# B&R Automation Studio project CombinedLinenSoiledA9KAN (part 15)

#### _actInterfaceApplication.st
```iecst
(********************************************************************
 * COPYRIGHT -- Herbert Kannegiesser GmbH
 ********************************************************************
 * Program: mnParam
 * File: _actInterfaceApplication.st
 * Author: hunholz
 * Created: March 28, 2012
 ********************************************************************
 * Implementation of program mnParam
 ********************************************************************)

(* Kommando-Interface zur Applikation über IFmnParam *)
ACTION _actInterfaceApplication:

	CASE _PmIntern.enCycIfState OF

		cs_IfIdle:

			//*************************************************
			// Kein Applikations-Befehl aktiv. Warte auf Befehl
			//*************************************************

			CASE IFmnParam.In.Edit.wCommand OF

				MNPARAM_CMD_NOCOMMAND:

					IFmnParam.Out.Edit.wStatus := MNPARAM_STAT_NOCOMMAND;

				MNPARAM_CMD_FILLEDITOR:

					IF _xAllowCommands THEN

						_xAllowCommands := FALSE;

						// Warten bis das Füllen des Editors abgeschlossen ist.
						_PmIntern.enCycIfState := cs_IfFillEditor;

						IFmnParam.Out.Edit.wStatus := KG_CMDSTAT_BUSY;

						// Füllen des Editors starten
						_PmIntern.enCycFillEditor := cs_feStart;

					ELSE

						// Kommando ablehnen
						IFmnParam.Out.Edit.wStatus := KG_CMDSTAT_NOTREADY;
						// Kommando muss zurückgenommen werden
						_PmIntern.enCycIfState := cs_IfReady;

					END_IF

				MNPARAM_CMD_SAVEEDITOR:

					IF _xAllowCommands THEN

						_xAllowCommands := FALSE;

						// Warten bis das Sichern des Editors abgeschlossen ist
						_PmIntern.enCycIfState := cs_IfSaveEditor;

						IFmnParam.Out.Edit.wStatus := KG_CMDSTAT_BUSY;

						_LogEntryIn.wErrorNo := _MNPARAM_LOG_STARTSAVE;
						_InsertRB(wPtrStart := _wPtrRBstart, wPtrRead := _wPtrRBread, wPtrWrite := _wPtrRBwrite);

						// Sichern starten
						_PmIntern.enCycSaveEditor := cs_seStart;

					ELSE

						// Kommando ablehnen
						IFmnParam.Out.Edit.wStatus := KG_CMDSTAT_NOTREADY;
						// Kommando muss zurückgenommen werden
						_PmIntern.enCycIfState := cs_IfReady;

					END_IF

				MNPARAM_CMD_CREATE_INDCONT:

					IF _xAllowCommands THEN

						_xAllowCommands := FALSE;

						// Warten bis das Anlegen einer Instanz abgeschlossen ist
						_PmIntern.enCycIfState := cs_IfCreateIndCont;

						IFmnParam.Out.Edit.wStatus := KG_CMDSTAT_BUSY;

						// Parameter übernehmen
						_wCreateCont := IFmnParam.In.Edit.bContainer;
						_wCreateInst := IFmnParam.In.Edit.wContainerInstance;

						_LogEntryIn.wErrorNo := _MNPARAM_LOG_STARTCREATE;
						_LogEntryIn.lAttr1 := _wCreateCont;
						_LogEntryIn.lAttr2 := _wCreateInst;
						_InsertRB(wPtrStart := _wPtrRBstart, wPtrRead := _wPtrRBread, wPtrWrite := _wPtrRBwrite);

						// Instanz anlegen
						_PmIntern.enCycCreate := cs_CrtStart;

					ELSE

						// Kommando ablehnen
						IFmnParam.Out.Edit.wStatus := KG_CMDSTAT_NOTREADY;
						// Kommando muss zurückgenommen werden
						_PmIntern.enCycIfState := cs_IfReady;

					END_IF

				MNPARAM_CMD_DELETE_INDCONT:

					IF _xAllowCommands THEN

						_xAllowCommands := FALSE;

						// Warten bis das Löschen der Instanz abgeschlossen ist
						_PmIntern.enCycIfState := cs_IfDeleteIndCont;

						IFmnParam.Out.Edit.wStatus := KG_CMDSTAT_BUSY;

						// Parameter übernehmen
						_wDelCont := IFmnParam.In.Edit.bContainer;
						_wDelInst := IFmnParam.In.Edit.wContainerInstance;

						_LogEntryIn.wErrorNo := _MNPARAM_LOG_STARTDELETE;
						_LogEntryIn.lAttr1 := _wDelCont;
						_LogEntryIn.lAttr2 := _wDelInst;
						_InsertRB(wPtrStart := _wPtrRBstart, wPtrRead := _wPtrRBread, wPtrWrite := _wPtrRBwrite);

						// Löschen starten
						_PmIntern.enCycDelState := cs_DelStart;

					ELSE

						// Kommando ablehnen
						IFmnParam.Out.Edit.wStatus := KG_CMDSTAT_NOTREADY;
						// Kommando muss zurückgenommen werden
						_PmIntern.enCycIfState := cs_IfReady;

					END_IF

				MNPARAM_CMD_COPY_INDCONT:

					IF _xAllowCommands THEN

						_xAllowCommands := FALSE;

						// Warten bis das Kopieren der Instanz abgeschlossen ist
						_PmIntern.enCycIfState := cs_IfCopyIndCont;

						IFmnParam.Out.Edit.wStatus := KG_CMDSTAT_BUSY;

						// Parameter übernehmen
						_wCopyCont := IFmnParam.In.Edit.bContainer;
						_wCopyInst := IFmnParam.In.Edit.wContainerInstance;
						_wCopyInstFrom := IFmnParam.In.Edit.wContainerInstanceFrom;

						_LogEntryIn.wErrorNo := _MNPARAM_LOG_STARTCOPY;
						_LogEntryIn.lAttr1 := _wCopyCont;
						_LogEntryIn.lAttr2 := _wCopyInst;
						_InsertRB(wPtrStart := _wPtrRBstart, wPtrRead := _wPtrRBread, wPtrWrite := _wPtrRBwrite);

						// Kopieren starten
						_PmIntern.enCycCopy := cs_CpyStart;

					ELSE

						// Kommando ablehnen
						IFmnParam.Out.Edit.wStatus := KG_CMDSTAT_NOTREADY;
						// Kommando muss zurückgenommen werden
						_PmIntern.enCycIfState := cs_IfReady;

					END_IF

				MNPARAM_CMD_BACKUP:

					IF _xAllowCommands THEN

						_xAllowCommands := FALSE;

						// USB-Flashdisk muss gesteckt sein
						IF IFmnSystem.Out.xUSBStickReady THEN

							// Warten bis Backup beendet ist
							_PmIntern.enCycIfState := cs_IfBackup;

							IFmnParam.Out.Edit.wStatus := KG_CMDSTAT_BUSY;

							_LogEntryIn.wErrorNo := _MNPARAM_LOG_STARTBACKUP;
							_LogEntryIn.lAttr1 := 0;
							_LogEntryIn.lAttr2 := 0;
							_InsertRB(wPtrStart := _wPtrRBstart, wPtrRead := _wPtrRBread, wPtrWrite := _wPtrRBwrite);

							// Devicenamen der USB-Flashdisk übernehmen
							_sUSBInterface := IFmnSystem.Out.sInterfaceUSB;

							// Backup starten
							_PmIntern.enCycBackup := cs_BacUSBlinkDevice;

						ELSE

							// Es ist keine USB-Flashdisk gesteckt
							IFmnParam.Out.Edit.wStatus := MNPARAM_STAT_NOUSBSTICK;
							// Kommando muss zurückgenommen werden
							_PmIntern.enCycIfState := cs_IfReady;

						END_IF

					ELSE

						// Kommando ablehnen
						IFmnParam.Out.Edit.wStatus := KG_CMDSTAT_NOTREADY;
						// Kommando muss zurückgenommen werden
						_PmIntern.enCycIfState := cs_IfReady;

					END_IF

				MNPARAM_CMD_RESTORE:

					IF _xAllowCommands THEN

						_xAllowCommands := FALSE;

						// USB-Flashdisk muss gesteckt sein
						IF IFmnSystem.Out.xUSBStickReady THEN

							// Warten bis Restore abgeschlossen ist
							_PmIntern.enCycIfState := cs_IfRestore;

							IFmnParam.Out.Edit.wStatus := KG_CMDSTAT_BUSY;

							// Devicenamen der USB-Flashdisk übernehmen
							_sUSBInterface := IFmnSystem.Out.sInterfaceUSB;

							_LogEntryIn.wErrorNo := _MNPARAM_LOG_STARTRESTORE;
							_LogEntryIn.lAttr1 := 0;
							_LogEntryIn.lAttr2 := 0;
							_InsertRB(wPtrStart := _wPtrRBstart, wPtrRead := _wPtrRBread, wPtrWrite := _wPtrRBwrite);

							// Restore starten
							_PmIntern.enCycImpState := cs_ImpUSBLinkDevice;

						ELSE

							// Es ist keine USB-Flashdisk gesteckt
							IFmnParam.Out.Edit.wStatus := MNPARAM_STAT_NOUSBSTICK;
							// Kommando muss zurückgenommen werden
							_PmIntern.enCycIfState := cs_IfReady;

						END_IF

					ELSE

						// Kommando ablehnen
						IFmnParam.Out.Edit.wStatus := KG_CMDSTAT_NOTREADY;
						// Kommando muss zurückgenommen werden
						_PmIntern.enCycIfState := cs_IfReady;

					END_IF

				MNPARAM_CMD_FILLNAMELIST:

					IF _xAllowCommands THEN

						_xAllowCommands := FALSE;

						IFmnParam.Out.Edit.wIdxContainerNamelist := IFmnParam.In.Edit.wSelIdxContainerNamelist;
						IFmnParam.Out.Edit.wParIdxNamelist := IFmnParam.In.Edit.wSelParIdxNamelist;

						_actFillNamelist;

						IFmnParam.Out.Edit.wStatus := MNPARAM_STAT_FILLNAMELIST_OK;

						_PmIntern.enCycIfState := cs_IfReady;

					END_IF

				ELSE

					// Kommando ungültig
					IFmnParam.Out.Edit.wStatus := KG_CMDSTAT_NOTVALID;
					// Kommando muss zurückgenommen werden
					_PmIntern.enCycIfState := cs_IfReady;

			END_CASE

		cs_IfFillEditor:

			// Warten bis Füllen des Editor fertig ist
			IF _PmIntern.enCycFillEditor = cs_feRdySuccess THEN

				// ERFOLG

				// Rückmeldung
				IFmnParam.Out.Edit.wStatus := MNPARAM_STAT_FILLEDITOR_OK;

				// Statemachine Editor Füllen zurücksetzen
				_PmIntern.enCycFillEditor := cs_feIdle;
				// Kommando muss zurückgenommen werden
				_PmIntern.enCycIfState := cs_IfReady;

			ELSIF _PmIntern.enCycFillEditor = cs_feRdyFault THEN

				// FEHLER

				// Status zurückliefern
				IFmnParam.Out.Edit.wStatus := DINT_TO_UINT(_PmIntern.Status.diMsgAttr1);

				// Statemachine Editor Füllen zurücksetzen
				_PmIntern.enCycFillEditor := cs_feIdle;
				// Kommando muss zurückgenommen werden
				_PmIntern.enCycIfState := cs_IfReady;

			END_IF

		cs_IfSaveEditor:

			// Warten bis Editor gesichert wurde
			IF _PmIntern.enCycSaveEditor = cs_seRdySuccess THEN

				// ERFOLG

				// Rückmeldung
				IFmnParam.Out.Edit.wStatus := MNPARAM_STAT_SAVEEDITOR_OK;

				// Statemchine Editor sichern zurücksetzen
				_PmIntern.enCycSaveEditor := cs_seIdle;
				// Kommando muss zurückgenommen werden
				_PmIntern.enCycIfState := cs_IfReady;

				_LogEntryIn.wErrorNo := _MNPARAM_LOG_ENDSAVE_SUCC;
				_InsertRB(wPtrStart := _wPtrRBstart, wPtrRead := _wPtrRBread, wPtrWrite := _wPtrRBwrite);

			ELSIF _PmIntern.enCycSaveEditor = cs_seRdyFault THEN

				// FEHLER

				// Status zurückmelden
				IFmnParam.Out.Edit.wStatus := DINT_TO_UINT(_PmIntern.Status.diMsgAttr1);

				// Statemchine Editor sichern zurücksetzen
				_PmIntern.enCycSaveEditor := cs_seIdle;
				// Kommando muss zurückgenommen werden
				_PmIntern.enCycIfState := cs_IfReady;

				_LogEntryIn.wErrorNo := _MNPARAM_LOG_ENDSAVE_FAILED;
				_LogEntryIn.lAttr1 := IFmnParam.Out.Edit.wStatus;
				_InsertRB(wPtrStart := _wPtrRBstart, wPtrRead := _wPtrRBread, wPtrWrite := _wPtrRBwrite);

			END_IF

		cs_IfCreateIndCont:

			// Warten bis Instanz angelegt wurde
			IF _PmIntern.enCycCreate = cs_CrtRdySuccess THEN

				// ERFOLG

				// Rückmeldung
				IFmnParam.Out.Edit.wStatus := MNPARAM_STAT_CREATE_INDCONT_OK;

				// Statemachine Instanz anlegen zurücksetzen
				_PmIntern.enCycCreate := cs_CrtIdle;
				// Kommando muss zurückgenommen werden
				_PmIntern.enCycIfState := cs_IfReady;

				_LogEntryIn.wErrorNo := _MNPARAM_LOG_ENDCREATE_SUCC;
				_InsertRB(wPtrStart := _wPtrRBstart, wPtrRead := _wPtrRBread, wPtrWrite := _wPtrRBwrite);

				IF _wCreateCont = MNPARAM_IDX_PROGCONTAINER THEN

					_actFillNamelist;

				END_IF

			ELSIF _PmIntern.enCycCreate = cs_CrtRdyFault THEN

				// FEHLER

				// Status zurückmelden
				IFmnParam.Out.Edit.wStatus := DINT_TO_UINT(_PmIntern.Status.diMsgAttr1);

				// Statemachine Instanz anlegen zurücksetzen
				_PmIntern.enCycCreate := cs_CrtIdle;
				// Kommando muss zurückgenommen werden
				_PmIntern.enCycIfState := cs_IfReady;

				_LogEntryIn.wErrorNo := _MNPARAM_LOG_ENDCREATE_FAILED;
				_LogEntryIn.lAttr1 := IFmnParam.Out.Edit.wStatus;
				_InsertRB(wPtrStart := _wPtrRBstart, wPtrRead := _wPtrRBread, wPtrWrite := _wPtrRBwrite);

			END_IF

		cs_IfDeleteIndCont:

			// Warten bis Instanz löschen fertig ist
			IF _PmIntern.enCycDelState = cs_DelRdySuccess THEN

				// ERFOLG

				// Rückmeldung
				IFmnParam.Out.Edit.wStatus := MNPARAM_STAT_DELETE_INDCONT_OK;

				// Statemachin Delete zurücksetzen
				_PmIntern.enCycDelState := cs_DelIdle;
				// Kommando muss zurückgenommen werden
				_PmIntern.enCycIfState := cs_IfReady;

				_LogEntryIn.wErrorNo := _MNPARAM_LOG_ENDDELETE_SUCC;
				_InsertRB(wPtrStart := _wPtrRBstart, wPtrRead := _wPtrRBread, wPtrWrite := _wPtrRBwrite);

				IF _wDelCont = MNPARAM_IDX_PROGCONTAINER THEN

					_actFillNamelist;

				END_IF

			ELSIF _PmIntern.enCycDelState = cs_DelRdyFault THEN

				// FEHLER

				// Status zurückmelden
				IFmnParam.Out.Edit.wStatus := MAX(59999,DINT_TO_UINT(_PmIntern.Status.diMsgAttr1));

				// Statemachin Delete zurücksetzen
				_PmIntern.enCycDelState := cs_DelIdle;
				// Kommando muss zurückgenommen werden
				_PmIntern.enCycIfState := cs_IfReady;

				_LogEntryIn.wErrorNo := _MNPARAM_LOG_ENDDELETE_FAILED;
				_LogEntryIn.lAttr1 := IFmnParam.Out.Edit.wStatus;
				_InsertRB(wPtrStart := _wPtrRBstart, wPtrRead := _wPtrRBread, wPtrWrite := _wPtrRBwrite);

			END_IF

		cs_IfCopyIndCont:

			// Warten bis Instanz kopiert wurde
			IF _PmIntern.enCycCopy = cs_CpyRdySuccess THEN

				// ERFOLG

				// Status zurückmelden
				IFmnParam.Out.Edit.wStatus := MNPARAM_STAT_COPY_INDCONT_OK;

				// Statemachine Kopieren zurücksetzen
				_PmIntern.enCycCopy := cs_CpyIdle;
				// Kommando muss zurückgenommen werden
				_PmIntern.enCycIfState := cs_IfReady;

				_LogEntryIn.wErrorNo := _MNPARAM_LOG_ENDCOPY_SUCC;
				_InsertRB(wPtrStart := _wPtrRBstart, wPtrRead := _wPtrRBread, wPtrWrite := _wPtrRBwrite);

				IF _wCopyCont = MNPARAM_IDX_PROGCONTAINER THEN

					_actFillNamelist;

				END_IF

			ELSIF _PmIntern.enCycCopy = cs_CpyRdyFault THEN

				// FEHLER

				// Status zurückmelden
				IFmnParam.Out.Edit.wStatus := DINT_TO_UINT(_PmIntern.Status.diMsgAttr1);

				// Statemachine Kopieren zurücksetzen
				_PmIntern.enCycCopy := cs_CpyIdle;
				// Kommando muss zurückgenommen werden
				_PmIntern.enCycIfState := cs_IfReady;

				_LogEntryIn.wErrorNo := _MNPARAM_LOG_ENDCOPY_FAILED;
				_LogEntryIn.lAttr1 := IFmnParam.Out.Edit.wStatus;
				_InsertRB(wPtrStart := _wPtrRBstart, wPtrRead := _wPtrRBread, wPtrWrite := _wPtrRBwrite);

			END_IF

		cs_IfBackup:

			// Warten bis Backup fertig ist
			IF _PmIntern.enCycBackup = cs_BacRdySuccess THEN

				// ERFOLG

				// Rückmeldung
				IFmnParam.Out.Edit.wStatus := MNPARAM_STAT_BACKUP_OK;

				// Statemachine Backup zurücksetzen
				_PmIntern.enCycBackup := cs_BacIdle;
				// Kommando muss zurückgenommen werden
				_PmIntern.enCycIfState := cs_IfReady;

				_LogEntryIn.wErrorNo := _MNPARAM_LOG_ENDBACKUP_SUCC;
				_InsertRB(wPtrStart := _wPtrRBstart, wPtrRead := _wPtrRBread, wPtrWrite := _wPtrRBwrite);

			ELSIF _PmIntern.enCycBackup = cs_BacRdyFault THEN

				// FEHLER

				// Status zurückmelden
				IFmnParam.Out.Edit.wStatus := MAX(59999,DINT_TO_UINT(_PmIntern.Status.diMsgAttr1));

				// Statemachine Backup zurücksetzen
				_PmIntern.enCycBackup := cs_BacIdle;
				// Kommando muss zurückgenommen werden
				_PmIntern.enCycIfState := cs_IfReady;

				_LogEntryIn.wErrorNo := _MNPARAM_LOG_ENDBACKUP_FAILED;
				_LogEntryIn.lAttr1 := IFmnParam.Out.Edit.wStatus;
				_InsertRB(wPtrStart := _wPtrRBstart, wPtrRead := _wPtrRBread, wPtrWrite := _wPtrRBwrite);

			END_IF

		cs_IfRestore:

			// Warten bis Import/Restore fertig ist
			IF _PmIntern.enCycImpState = cs_ImpRdySuccess THEN

				// ERFOLGE

				// Rückmeldung
				IFmnParam.Out.Edit.wStatus := MNPARAM_STAT_RESTORE_OK;

				// Statemachine Import zurücksetzen
				_PmIntern.enCycImpState := cs_ImpIdle;
				// Kommando muss zurückgenommen werden
				_PmIntern.enCycIfState := cs_IfReady;

				_LogEntryIn.wErrorNo := _MNPARAM_LOG_ENDRESTORE_SUCC;
				_InsertRB(wPtrStart := _wPtrRBstart, wPtrRead := _wPtrRBread, wPtrWrite := _wPtrRBwrite);

				_actFillNamelist;

			ELSIF _PmIntern.enCycImpState = cs_ImpRdyFault THEN

				// FEHLER

				// Status zurückmelden
				IFmnParam.Out.Edit.wStatus := MAX(59999,DINT_TO_UINT(_PmIntern.Status.diMsgAttr1));

				// Statemachine Import zurücksetzen
				_PmIntern.enCycImpState := cs_ImpIdle;
				// Kommando muss zurückgenommen werden
				_PmIntern.enCycIfState := cs_IfReady;

				_LogEntryIn.wErrorNo := _MNPARAM_LOG_ENDRESTORE_FAILED;
				_LogEntryIn.lAttr1 := IFmnParam.Out.Edit.wStatus;
				_InsertRB(wPtrStart := _wPtrRBstart, wPtrRead := _wPtrRBread, wPtrWrite := _wPtrRBwrite);

			END_IF

		cs_IfReady:

			// Warten, bis das Kommando zurückgenommen wurde. Bei Warnung mindestzeit abwarten
			IF IFmnParam.In.Edit.wCommand = MNPARAM_CMD_NOCOMMAND AND (_PmIntern.Status.wMsgNumber = 0 OR TONwarn2.Q) THEN

				// Rückmeldung
				IFmnParam.Out.Edit.wStatus := MNPARAM_STAT_NOCOMMAND;

				// Meldung zurücksetzen
				brsmemset(ADR(_PmIntern.Status), 0, SIZEOF(_PmIntern.Status));
				_PmIntern.Status.wFunction_ID := MNPARAM_FUNCTIONID;

				// Interface zur Applikation wieder bereit schalten
				_PmIntern.enCycIfState := cs_IfIdle;

			END_IF

	END_CASE

	// Warnung soll mindestens 4 Sekunden anstehen
	TONwarn2(IN := _PmIntern.enCycIfState = cs_IfReady, PT := T#4s);

END_ACTION
```

#### _actFillEditNum.st
```iecst
(********************************************************************
 * COPYRIGHT -- Herbert Kannegiesser GmbH
 ********************************************************************
 * Program: mnParam
 * File: _actFillEditNum.st
 * Author: hunholz
 * Created: March 21, 2012
 ********************************************************************
 * Implementation of program mnParam
 ********************************************************************)

(* Attribute und Werte füllen *)
ACTION _actFillEditNum:

	// Attribute übertragen

	IFmnParam.Out.Edit.AttrNum[_wActRow].wType := _pDoParamNum.ParamNum[_wActRefIdx].bRowType + MNPARAM_CSV_DAT_NUM;
	IFmnParam.Out.Edit.AttrNum[_wActRow].wUnit := _pDoParamNum.ParamNum[_wActRefIdx].wUnitID;
	IFmnParam.Out.Edit.AttrNum[_wActRow].wFunctionID := _pDoParamNum.ParamNum[_wActRefIdx].wFunction_ID;
	IFmnParam.Out.Edit.AttrNum[_wActRow].wParamNo := _pDoParamNum.ParamNum[_wActRefIdx].wParNo;
	IFmnParam.Out.Edit.AttrNum[_wActRow].wParIdx := _wActRefIdx;
	IFmnParam.Out.Edit.AttrNum[_wActRow].wArrIdx[1] := _pDoContainerNum.CsvNum[_wActIdx].wArrIdx1;
	IFmnParam.Out.Edit.AttrNum[_wActRow].wArrIdx[2] := _pDoContainerNum.CsvNum[_wActIdx].wArrIdx2;
	IFmnParam.Out.Edit.AttrNum[_wActRow].wArrIdx[3] := _pDoContainerNum.CsvNum[_wActIdx].wArrIdx3;
	IFmnParam.Out.Edit.AttrNum[_wActRow].wArrIdx[4] := _pDoContainerNum.CsvNum[_wActIdx].wArrIdx4;

	_pDigits := ADR(IFmnParam.Out.Edit.AttrNum[_wActRow].lDigits);
	_pUnit := ADR(IFmnParam.Out.Edit.AttrNum[_wActRow].sUnit);

	IF _pDoParamNum.ParamNum[_wActRefIdx].bRowType = 0 THEN

		// INT
		IFmnParam.Out.Edit.AttrNum[_wActRow].rDefault := kgUnitconfREALtoDisplay(DINT_TO_REAL(_pDoParamNum.ParamNum[_wActRefIdx].diDefValue),_pDoParamNum.ParamNum[_wActRefIdx].wUnitID,IFmnParam.In.Edit.bLocUnit, _pDigits, _pUnit);
		IFmnParam.Out.Edit.AttrNum[_wActRow].rMax := kgUnitconfREALtoDisplay(DINT_TO_REAL(_pDoParamNum.ParamNum[_wActRefIdx].diMaxValue),_pDoParamNum.ParamNum[_wActRefIdx].wUnitID,IFmnParam.In.Edit.bLocUnit, 0, 0);
		IFmnParam.Out.Edit.AttrNum[_wActRow].rMin := kgUnitconfREALtoDisplay(DINT_TO_REAL(_pDoParamNum.ParamNum[_wActRefIdx].diMinValue),_pDoParamNum.ParamNum[_wActRefIdx].wUnitID,IFmnParam.In.Edit.bLocUnit, 0, 0);

	ELSE

		// REAL
		_prValue ACCESS ADR(_pDoParamNum.ParamNum[_wActRefIdx].diDefValue);
		IFmnParam.Out.Edit.AttrNum[_wActRow].rDefault := kgUnitconfREALtoDisplay(_prValue,_pDoParamNum.ParamNum[_wActRefIdx].wUnitID,IFmnParam.In.Edit.bLocUnit, _pDigits, _pUnit);
		_prValue ACCESS ADR(_pDoParamNum.ParamNum[_wActRefIdx].diMaxValue);
		IFmnParam.Out.Edit.AttrNum[_wActRow].rMax := kgUnitconfREALtoDisplay(_prValue,_pDoParamNum.ParamNum[_wActRefIdx].wUnitID,IFmnParam.In.Edit.bLocUnit, 0, 0);
		_prValue ACCESS ADR(_pDoParamNum.ParamNum[_wActRefIdx].diMinValue);
		IFmnParam.Out.Edit.AttrNum[_wActRow].rMin := kgUnitconfREALtoDisplay(_prValue,_pDoParamNum.ParamNum[_wActRefIdx].wUnitID,IFmnParam.In.Edit.bLocUnit, 0, 0);

	END_IF

	// Wert übergeben

	IF _pDoParamNum.ParamNum[_wActRefIdx].bRowType = 0 THEN
		_EditNumValues.rVal[_wActRow] := kgUnitconfREALtoDisplay(DINT_TO_REAL(_pDoContainerNum.CsvNum[_wActIdx].diValue),_pDoParamNum.ParamNum[_wActRefIdx].wUnitID,IFmnParam.In.Edit.bLocUnit, 0, 0);
	ELSE
		_prValue ACCESS ADR(_pDoContainerNum.CsvNum[_wActIdx].diValue);
		_EditNumValues.rVal[_wActRow] := kgUnitconfREALtoDisplay(_prValue,_pDoParamNum.ParamNum[_wActRefIdx].wUnitID,IFmnParam.In.Edit.bLocUnit, 0, 0);
	END_IF

	_EditNumValues.wIdx[_wActRow] := _wActIdx;

	// Texte übergeben (Binäre Suche)

	IF IFmnTxt.Out.wSelectLanguageStatus = ERR_OK AND IFmnTxt.Out.ptrFunctionTxtList <> 0 AND IFmnTxt.Out.ptrInstanceTxtList <> 0 AND

		IFmnTxt.Out.ptrParamTxtList <> 0 AND IFmnTxt.Out.ptrParamHelpTxtList <> 0 THEN

		_wIdxFunctionTxt := _BinSearchTxtLine(IFmnParam.Out.Edit.AttrNum[_wActRow].wFunctionID, 0, IFmnTxt.Out.ptrFunctionTxtList, IFmnTxt.Out.wCntFunctionTxt);

		_wIdxInstanceTxt := _BinSearchTxtLine(IFmnParam.Out.Edit.AttrNum[_wActRow].wFunctionID, IFmnParam.Out.Edit.AttrNum[_wActRow].wArrIdx[1],
		IFmnTxt.Out.ptrInstanceTxtList, IFmnTxt.Out.wCntInstanceTxt);

		_wIdxParamTxt := _BinSearchTxtLine(IFmnParam.Out.Edit.AttrNum[_wActRow].wFunctionID, IFmnParam.Out.Edit.AttrNum[_wActRow].wParamNo,
		IFmnTxt.Out.ptrParamTxtList, IFmnTxt.Out.wCntParamTxt);

		_wIdxParamHlpTxt := _BinSearchHlpTxtLine(IFmnParam.Out.Edit.AttrNum[_wActRow].wFunctionID, IFmnParam.Out.Edit.AttrNum[_wActRow].wParamNo,
		IFmnTxt.Out.ptrParamHelpTxtList, IFmnTxt.Out.wCntParamHlpTxt);

		IFmnParam.Out.Edit.AttrNum[_wActRow].utfParameterName := "";
		IFmnParam.Out.Edit.AttrNum[_wActRow].utfParameterHelpTxt := "";
		_wLenUtf := 0;

		IF _wIdxFunctionTxt <> 65535 THEN
			_pFunctionTxt ACCESS IFmnTxt.Out.ptrFunctionTxtList;
			brwcsncat(ADR(IFmnParam.Out.Edit.AttrNum[_wActRow].utfParameterName), ADR(_pFunctionTxt[_wIdxFunctionTxt].utfText), 63-_wLenUtf);
			_wLenUtf := UDINT_TO_UINT(brwcslen(ADR(IFmnParam.Out.Edit.AttrNum[_wActRow].utfParameterName)));
			brwcsncat(ADR(IFmnParam.Out.Edit.AttrNum[_wActRow].utfParameterName), ADR("."), 63-_wLenUtf);
			_wLenUtf := UDINT_TO_UINT(brwcslen(ADR(IFmnParam.Out.Edit.AttrNum[_wActRow].utfParameterName)));
		END_IF

		IF _wIdxInstanceTxt <> 65535 THEN
			_pInstanceTxt ACCESS IFmnTxt.Out.ptrInstanceTxtList;
			brwcsncat(ADR(IFmnParam.Out.Edit.AttrNum[_wActRow].utfParameterName), ADR(_pInstanceTxt[_wIdxInstanceTxt].utfText), 63-_wLenUtf);
			_wLenUtf := UDINT_TO_UINT(brwcslen(ADR(IFmnParam.Out.Edit.AttrNum[_wActRow].utfParameterName)));
			brwcsncat(ADR(IFmnParam.Out.Edit.AttrNum[_wActRow].utfParameterName), ADR("."), 63-_wLenUtf);
			_wLenUtf := UDINT_TO_UINT(brwcslen(ADR(IFmnParam.Out.Edit.AttrNum[_wActRow].utfParameterName)));
		END_IF

		IF _wIdxParamTxt <> 65535 THEN
			_pParamTxt ACCESS IFmnTxt.Out.ptrParamTxtList;
			brwcsncat(ADR(IFmnParam.Out.Edit.AttrNum[_wActRow].utfParameterName), ADR(_pParamTxt[_wIdxParamTxt].utfText), 63-_wLenUtf);
		END_IF

		IF _wIdxParamHlpTxt <> 65535 THEN
			_pParamHlpTxt ACCESS IFmnTxt.Out.ptrParamHelpTxtList;
			brwcsncat(ADR(IFmnParam.Out.Edit.AttrNum[_wActRow].utfParameterHelpTxt), ADR(_pParamHlpTxt[_wIdxParamHlpTxt].utfText), 63);
		END_IF

	END_IF

END_ACTION
```

#### _actFillEditStr.st
```iecst
(********************************************************************
 * COPYRIGHT -- Herbert Kannegiesser GmbH
 ********************************************************************
 * Program: mnParam
 * File: _actFillEditStr.st
 * Author: hunholz
 * Created: March 21, 2012
 ********************************************************************
 * Implementation of program mnParam
 ********************************************************************)

(* Attribute und Werte *)
ACTION _actFillEditStr:

	// Attribute übertragen

	IFmnParam.Out.Edit.AttrStr[_wActRow].wType := 20;
	IFmnParam.Out.Edit.AttrStr[_wActRow].wFunctionID := _pDoParamString.ParamString[_wActRefIdx].wFunction_ID;
	IFmnParam.Out.Edit.AttrStr[_wActRow].wParamNo := _pDoParamString.ParamString[_wActRefIdx].wParNo;
	IFmnParam.Out.Edit.AttrStr[_wActRow].wParIdx := _wActRefIdx;
	IFmnParam.Out.Edit.AttrStr[_wActRow].wArrIdx[1] := _pDoContainerString.CsvString[_wActIdx].wArrIdx1;
	IFmnParam.Out.Edit.AttrStr[_wActRow].wArrIdx[2] := _pDoContainerString.CsvString[_wActIdx].wArrIdx2;
	IFmnParam.Out.Edit.AttrStr[_wActRow].wArrIdx[3] := _pDoContainerString.CsvString[_wActIdx].wArrIdx3;
	IFmnParam.Out.Edit.AttrStr[_wActRow].wArrIdx[4] := _pDoContainerString.CsvString[_wActIdx].wArrIdx4;

	IFmnParam.Out.Edit.AttrStr[_wActRow].utfDefault := _pDoParamString.ParamString[_wActRefIdx].utfDefValue;
	IFmnParam.Out.Edit.AttrStr[_wActRow].wMaxLength := _pDoParamString.ParamString[_wActRefIdx].bLenght;

	// Wert übergeben

	_EditStrValues.utfVal[_wActRow] := _pDoContainerString.CsvString[_wActIdx].utfValue;
	_EditStrValues.xSave[_wActRow] := FALSE;
	_EditStrValues.wIdx[_wActRow] := _wActIdx;

	// Texte übergeben (Binäre Suche)

	IF IFmnTxt.Out.wSelectLanguageStatus = ERR_OK AND IFmnTxt.Out.ptrFunctionTxtList <> 0 AND IFmnTxt.Out.ptrInstanceTxtList <> 0 AND
		IFmnTxt.Out.ptrParamTxtList <> 0 AND IFmnTxt.Out.ptrParamHelpTxtList <> 0 THEN

		_wIdxFunctionTxt := _BinSearchTxtLine(IFmnParam.Out.Edit.AttrStr[_wActRow].wFunctionID, 0, IFmnTxt.Out.ptrFunctionTxtList, IFmnTxt.Out.wCntFunctionTxt);

		_wIdxInstanceTxt := _BinSearchTxtLine(IFmnParam.Out.Edit.AttrStr[_wActRow].wFunctionID, IFmnParam.Out.Edit.AttrStr[_wActRow].wArrIdx[1],
		IFmnTxt.Out.ptrInstanceTxtList, IFmnTxt.Out.wCntInstanceTxt);

		_wIdxParamTxt := _BinSearchTxtLine(IFmnParam.Out.Edit.AttrStr[_wActRow].wFunctionID, IFmnParam.Out.Edit.AttrStr[_wActRow].wParamNo,
		IFmnTxt.Out.ptrParamTxtList, IFmnTxt.Out.wCntParamTxt);

		_wIdxParamHlpTxt := _BinSearchHlpTxtLine(IFmnParam.Out.Edit.AttrStr[_wActRow].wFunctionID, IFmnParam.Out.Edit.AttrStr[_wActRow].wParamNo,
		IFmnTxt.Out.ptrParamHelpTxtList, IFmnTxt.Out.wCntParamHlpTxt);

		IFmnParam.Out.Edit.AttrStr[_wActRow].utfParameterName := "";
		IFmnParam.Out.Edit.AttrStr[_wActRow].utfParameterHelpTxt := "";
		_wLenUtf := 0;

		IF _wIdxFunctionTxt <> 65535 THEN
			_pFunctionTxt ACCESS IFmnTxt.Out.ptrFunctionTxtList;
			brwcsncat(ADR(IFmnParam.Out.Edit.AttrStr[_wActRow].utfParameterName), ADR(_pFunctionTxt[_wIdxFunctionTxt].utfText), 63-_wLenUtf);
			_wLenUtf := UDINT_TO_UINT(brwcslen(ADR(IFmnParam.Out.Edit.AttrStr[_wActRow].utfParameterName)));
			brwcsncat(ADR(IFmnParam.Out.Edit.AttrStr[_wActRow].utfParameterName), ADR("."), 63-_wLenUtf);
			_wLenUtf := UDINT_TO_UINT(brwcslen(ADR(IFmnParam.Out.Edit.AttrStr[_wActRow].utfParameterName)));
		END_IF

		IF _wIdxInstanceTxt <> 65535 THEN
			_pInstanceTxt ACCESS IFmnTxt.Out.ptrInstanceTxtList;
			brwcsncat(ADR(IFmnParam.Out.Edit.AttrStr[_wActRow].utfParameterName), ADR(_pInstanceTxt[_wIdxInstanceTxt].utfText), 63-_wLenUtf);
			_wLenUtf := UDINT_TO_UINT(brwcslen(ADR(IFmnParam.Out.Edit.AttrStr[_wActRow].utfParameterName)));
			brwcsncat(ADR(IFmnParam.Out.Edit.AttrStr[_wActRow].utfParameterName), ADR("."), 63-_wLenUtf);
			_wLenUtf := UDINT_TO_UINT(brwcslen(ADR(IFmnParam.Out.Edit.AttrStr[_wActRow].utfParameterName)));
		END_IF

		IF _wIdxParamTxt <> 65535 THEN
			_pParamTxt ACCESS IFmnTxt.Out.ptrParamTxtList;
			brwcsncat(ADR(IFmnParam.Out.Edit.AttrStr[_wActRow].utfParameterName), ADR(_pParamTxt[_wIdxParamTxt].utfText), 63-_wLenUtf);
		END_IF

		IF _wIdxParamHlpTxt <> 65535 THEN
			_pParamHlpTxt ACCESS IFmnTxt.Out.ptrParamHelpTxtList;
			brwcsncat(ADR(IFmnParam.Out.Edit.AttrStr[_wActRow].utfParameterHelpTxt), ADR(_pParamHlpTxt[_wIdxParamHlpTxt].utfText), 63);
		END_IF

	END_IF

END_ACTION
```

### Library Logical/Mewa/KGFramework/Pkg_mnParam/mnParamLib (IEC)
Depends on: astime

### history.Pkg_mnParam.txt
```
0.2.0	18.8.2011	- Import-Verzeichnis wird im Hochlauf gelöscht
			- Es werden auch REAL-Parameter unterstützt. (not tested)
0.3.0	24.8.2011	- IP-CSV-Rowtype ergänzt. (90)
0.4.0	01.09.2011	- Info_typ geändert. Es wird jetzt auch ausgegeben, welcher Container geändert wurde
0.5.0	20.09.2011	- mnParamStat und mnParamStatAd ergänzt.
			  Kapselung von Stati. z.B. xParamOK, dtExportContent
0.6.0	07.10.2011	- Maschinennummer wird aus _mnr.csv gelesen und in die _Info_-Struktur geschrieben
0.6.1	18.11.2011	- Liefert jetzt eine Fehlermeldung, wenn die zu importierende Datei keine Maschinennummer enthält
0.6.2	28.11.2011	- mnParamLib : mnParam_WritePVNum. UDINT wurde als UINT behandelt.
0.7.0	20.10.2011	- Umstellung auf AS 3.0.90
					- Berücksichtigung von WSTRING
					- utfMachineNumber und xParamOK in das IFmnParam.Out
0.8.0	20.12.2011	- Logging in das Logbuch der AR verlegt.
					- EXIT hinzugefügt.
					- Fehler im Init-Up behoben.
0.8.1	22.12.2011	- Severity für Log angepasst
0.8.2	02.01.2012	- Initialisierung der Text-Zeilen in GetCsvDat
					- Sprachdefinition ist 248, nicht 247
0.9.0	03.01.2012	- Packetversion in mnParamStatAd
0.9.1	10.01.2012	- Kommentar der Package-Version im Export wird dynamisch gelesen
0.10.0	18.01.2012	- Textzeilen werden jetzt mit bis zu 63 Zeichen ausgelesen
0.11.0	13.02.2012	- Speicherloch in der Initialisierung beseitigt. Beim Importieren vorhandener Datencontainer wurde Speicher nicht mehr frei gegeben.
0.11.1	15.02.2012	- Weiterentwicklung: Speicheroptimierung. Automatische Berechnung der Größe der Speicherpartition.
		16.02.2012	- Einführung von Funktionsbausteinen für Standardfunktionen.
					- Schreiben eines Inhaltsverzeichnisses von CSV-Datencontainerdateien im Exportverzeichnis
		17.02.2012	- Unit ist UINT
0.11.2	22.02.2012	- Helptext wurde auf 63 Zeichen begrenzt
					- Kompatibel zu hlKanLink 0.94.0
0.12.0	06.03.2012	- Kompatibel zu mnTest
0.12.1	08.03.2012	- Bugfix Editliste füllen
0.13.0	15.03.2012	- Editliste wird mit umgerechneten Werten gefüllt.
0.13.1	15.03.2012	- Ergänzt um die Anzahl der Nachkommastellen
					- Datenmodell erweitert um RefVisible und RefText
0.13.2	20.03.2012	- Abhängigkeiten ergänzt
0.13.9	20.03.2012	- Zwischenstand - Weiterentwicklung mnParam
0.14.0	21.03.2012	- Save-Editor und Delete indirect container implementiert. Bugfix im Delete Algorithmus auch für mnParamCmd
0.15.0	22.03.2012	- Zwischenversion. Es wird jetzt für das Edit-Feld nach Parameterindex, und nicht nach Container-Index gesucht.
					- Letzter Parameter eines Containers wurde nicht ausgelesen
					- Massenimport implementiert
					- Restore ist möglich
0.15.1	23.03.2012	- Maschinennummer des Datencontainers wird jetzt auch im Init-Up überprüft.
					- Die Überprüfung der Maschinennummer im zyklischen Teil kann applikativ deaktiviert werden.
					- Logger implementiert
					- Backup und Restore implementiert
0.16.0	23.03.2012	- Release
0.16.1	27.03.2012	- Bugfix: Container wurden im Init-Up nicht eingelesen
0.16.2	27.03.2012	- Weiterentwicklung
0.17.0	28.03.2012	- Namensliste für Instanzen kann gefüllt werden
					- Instanz NEU und KOPIEREN ist implementiert
0.17.1	29.03.2012	- Bugfix. Save Editor. Letzter Eintrag wurde nicht gesichert
0.18.0	29.03.2012	- Kategorie-Programm-Zuordnung ergänzt
0.18.1	30.03.2012	- Kategorie-Programm-Zuordnung um Kategorienamen erweitert
0.18.2	02.04.2012	- Kategoriedaten erweitert
0.19.0	03.04.2012	- Warnungen bei Importfehler
		04.04.2012	- _Info_ wird nicht mehr unterstützt
					- Bugfix: TOC wurde beim Import vom PC nicht aktualisiert
0.20.0	05.04.2012	- Die Quelle zum Füllen der Namensliste wird nur initial von den Konstanten übernommen.
					  Per Befehl kann die Quelle geändert werden.
0.20.1	10.04.2012	- Wenn die Dateien im Exportverzeichnis gelöscht wurden, hat der Parametermanager diese nicht
					  neu angelegt.
0.20.2	11.04.2012	- Maschinennummer mit Länge 0 wird als Fehler abgefangen
0.20.3	11.04.2012	- Ungültige Maschinennummer "dummy" als Konstante MNPARAM_INVALID_MACHINENO eingeführt
0.20.4	13.04.2012	- Warnung wird angezeigt, wenn der Parametermanager nicht bereit ist.
0.20.5	16.04.2012	- Beim Füllen des Editors, wurden die Parameter für die Namensliste zurückgesetzt
0.20.6	17.04.2012	- Es konnten keine Instanzen aus dem Editor gesichert werden. Der Pointer auf die StrucRoot wurde nicht ermittelt.
0.20.7	18.04.2012  - Instanz-Datenobjekte werden im Init teilweise wieder gelöscht.
					- In der Instanznamensliste werden noch die Instanznummern vorangestellt
```

### Package Logical/Mewa/KGFramework/Pkg_mnTxt - Text-Manager

### Program Logical/Mewa/KGFramework/Pkg_mnTxt/mnTxt (IEC) - Text-Manager

#### mnTxtCyclic.st - Cyclic code
```iecst
(********************************************************************
 * COPYRIGHT -- Herbert Kannegiesser GmbH
 ********************************************************************
 * Program: mnTxt
 * File: mnTxtCyclic.st
 * Author: hunholz
 * Created: November 25, 2011
 ********************************************************************
 * Implementation of program mnTxt
 ********************************************************************)

PROGRAM _CYCLIC

	// Auf Sprachwechsel reagieren, bzw. letzte Sprache laden

	IF _xInitOK THEN

		IF IFmnTxt.Out.wSelectLanguageStatus = MNTXT_STAT_OK THEN

			// Sprache kann neu gewählt werden
			IF _wActLCID <> IFmnTxt.In.wSelectLanguage AND IFmnTxt.In.wSelectLanguage <> 0 THEN

				_wIdxLCID := 0;

				REPEAT

					IF IFmnTxt.In.wSelectLanguage = IFmnTxt.Out.wLCIDs[_wIdxLCID] THEN

						_wActLCID := IFmnTxt.In.wSelectLanguage;

						IFmnTxt.Out.wSelectedLanguage := _wActLCID;
						IFmnTxt.Out.wSelectLanguageStatus := MNTXT_STAT_LOADING;
						_LoadState := _ls_load_functiontxt_01;

					END_IF

					_wIdxLCID := _wIdxLCID + 1;

					UNTIL
					_wActLCID = IFmnTxt.In.wSelectLanguage OR _wIdxLCID >= IFmnTxt.Out.wCntLCID OR _wIdxLCID > MNTXT_MAX_IDX_LCID
				END_REPEAT

			END_IF

		ELSIF IFmnTxt.Out.wSelectLanguageStatus = MNTXT_STAT_NOLANGUAGE THEN

			IF _LoadState = _ls_idle THEN

				// Sprache erstmals laden
				IF _wActLCID = 0 THEN

					IF _xGermanExist THEN

						_wActLCID := MNTXT_LCID_GERMAN;

					ELSE

						_wActLCID := IFmnTxt.Out.wLCIDs[0];

					END_IF

				END_IF

				IFmnTxt.Out.wSelectedLanguage := _wActLCID;
				IFmnTxt.Out.wSelectLanguageStatus := MNTXT_STAT_LOADING;
				_LoadState := _ls_load_functiontxt_01;

			END_IF

		END_IF

	END_IF

	// Zyklusbegrenzung zurücksetzen

	_lCycleCounter := 0;

	// Statemachine

	CASE _LoadState OF

		_ls_idle:

		// Grundzustand, nichts tun

		//###########################################################################################
		// FUNKTIONSTEXTE LADEN
		//###########################################################################################

		_ls_load_functiontxt_01:

			// Nachsehen, ob Funktionstexte existieren

			IFmnTxt.Out.wCntFunctionTxt := 0;

			IF MNTXT_LOAD_FUNCTIONTEXT AND _CheckDoFunc.doId <> 0 THEN

				_FileInfo(enable := TRUE, pDevice := ADR(KG_DEVICE_COMPACTFLASH), pName := ADR('Language\Function.csv'), pInfo := ADR(_fiFileInfo));

				IF _FileInfo.status = ERR_OK THEN

					_LoadState := _ls_load_functiontxt_02;

				ELSIF _FileInfo.status <> ERR_FUB_BUSY THEN

					_LoadState := _ls_load_instancetxt_01;

				END_IF

			ELSE

				_LoadState := _ls_load_instancetxt_01;

			END_IF

		_ls_load_functiontxt_02:

			// Speicher zum Parsen der Funktionstexte allokieren
			_MemPartAlloc(enable := TRUE, ident := _MemPartCreate.ident, len := _fiFileInfo.size-SIZEOF(KGBOM) );

			IF _MemPartAlloc.status = ERR_OK THEN

				_lAdrFile := _MemPartAlloc.mem;
				_LoadState := _ls_load_functiontxt_03;

			ELSIF _MemPartAlloc.status <> ERR_FUB_BUSY THEN

				IFmnTxt.Out.wSelectLanguageStatus := MNTXT_STAT_ERRMEM;
				_LoadState := _ls_error;

			END_IF

		_ls_load_functiontxt_03:

			_FileOpen(enable := TRUE, pDevice := ADR(KG_DEVICE_COMPACTFLASH), pFile := ADR('Language\Function.csv'), mode := fiREAD_ONLY);

			IF _FileOpen.status = ERR_OK THEN

				_LoadState := _ls_load_functiontxt_04;

			ELSIF _FileOpen.status <> ERR_FUB_BUSY THEN

				IFmnTxt.Out.wSelectLanguageStatus := MNTXT_STAT_ERRFUNCTIONTXT;
				_LoadState := _ls_error;

			END_IF

		_ls_load_functiontxt_04:

			_FileRead(enable := TRUE, ident := _FileOpen.ident, offset := SIZEOF(KGBOM),pDest := _lAdrFile, len :=  _fiFileInfo.size-SIZEOF(KGBOM) );

			IF _FileRead.status <> ERR_FUB_BUSY THEN

				_LoadState := _ls_load_functiontxt_05;

			END_IF

		_ls_load_functiontxt_05:

			_FileClose(enable := TRUE, ident := _FileOpen.ident);

			IF _FileClose.status <> ERR_FUB_BUSY THEN

				IF _FileRead.status = ERR_OK THEN

					_LoadState := _ls_load_functiontxt_06;

				ELSE
					IFmnTxt.Out.wSelectLanguageStatus := MNTXT_STAT_ERRFUNCTIONTXT;
					_LoadState := _ls_error;

				END_IF

			END_IF

		_ls_load_functiontxt_06:

			// Zeilen in der Datei zählen und Startadressen ermitteln

			_CountLines.enable := TRUE;
			_CountLines.pFile := _lAdrFile;
			_CountLines.FileSize := _fiFileInfo.size - SIZEOF(KGBOM);
			_CountLines.MaxLines := MNTXT_MAXPARSELINES;
			_CountLines.pAdresses := _lAdrLineAdress;
			_CountLines.pLens := _lAdrLineLen;

			_CountLines();

			IF _CountLines.status = ERR_OK THEN

				_LoadState := _ls_load_functiontxt_07;

				_wStartLine := 1;
				_wIdxFunctionTxt := 0;
				_GetCsvDat.enable := TRUE;

			ELSE

				IFmnTxt.Out.wSelectLanguageStatus := MNTXT_STAT_ERRFUNCTIONTXT;
				_LoadState := _ls_error;

			END_IF

		_ls_load_functiontxt_07:

			// Datei parsen

			REPEAT

				brwcsncpy( ADR(_GetCsvDat.utfCsvString), _plLineAdress[_wStartLine], MIN(299, _pwLineLen[_wStartLine]));
				_GetCsvDat();
				_wStartLine := _wStartLine + 1;

				IF _GetCsvDat.RowType = 200 AND _GetCsvDat.csvTextRow.LCID = _wActLCID THEN

					_TxtLine.wNumber := 0;
					_TxtLine.wFunctionID := _GetCsvDat.csvTextRow.FunctionID;
					_TxtLine.utfText := _GetCsvDat.csvTextRow.utfText;

					_dowFuncTxt(enable := TRUE, ident := _CheckDoFunc.doId, Offset := SIZEOF(_TxtLine)*_wIdxFunctionTxt, pSource := ADR(_TxtLine), len := SIZEOF(_TxtLine));

					_wIdxFunctionTxt := _wIdxFunctionTxt + 1;

				END_IF

				_lCycleCounter := _lCycleCounter + 1;

				UNTIL

				_lCycleCounter > 20 OR _wIdxFunctionTxt > MNTXT_MAX_IDX_TXT_FUNCTION OR _wStartLine > _CountLines.CntLines

			END_REPEAT

			IF _wIdxFunctionTxt > MNTXT_MAX_IDX_TXT_FUNCTION OR _wStartLine > _CountLines.CntLines THEN

				IFmnTxt.Out.wCntFunctionTxt := _wIdxFunctionTxt;
				_LoadState := _ls_load_functiontxt_08;

			END_IF

		_ls_load_functiontxt_08:

			// Speicher frei geben

			_MemPartFree(enable := TRUE, ident := _MemPartCreate.ident, mem := _lAdrFile);

			IF _MemPartFree.status = ERR_OK THEN

				_LoadState := _ls_load_instancetxt_01;

			ELSIF _MemPartFree.status <> ERR_FUB_BUSY THEN

				IFmnTxt.Out.wSelectLanguageStatus := MNTXT_STAT_ERRFUNCTIONTXT;
				_LoadState := _ls_error;

			END_IF

		//###########################################################################################
		// INSTANZTEXTE LADEN
		//###########################################################################################

		_ls_load_instancetxt_01:

			// Nachsehen, ob Instanztexte existieren

			IFmnTxt.Out.wCntInstanceTxt := 0;

			IF MNTXT_LOAD_INSTANCETEXT AND _CheckDoInst.doId <> 0 THEN

				_FileInfo(enable := TRUE, pDevice := ADR(KG_DEVICE_COMPACTFLASH), pName := ADR('Language\Instance.csv'), pInfo := ADR(_fiFileInfo));

				IF _FileInfo.status = ERR_OK THEN

					_LoadState := _ls_load_instancetxt_02;

				ELSIF _FileInfo.status <> ERR_FUB_BUSY THEN

					_LoadState := _ls_load_messagetxt_01;

				END_IF

			ELSE

				_LoadState := _ls_load_messagetxt_01;

			END_IF

		_ls_load_instancetxt_02:

			// Speicher zum Parsen der Funktionstexte allokieren
			_MemPartAlloc(enable := TRUE, ident := _MemPartCreate.ident, len := _fiFileInfo.size-SIZEOF(KGBOM) );

			IF _MemPartAlloc.status = ERR_OK THEN

				_lAdrFile := _MemPartAlloc.mem;
				_LoadState := _ls_load_instancetxt_03;

			ELSIF _MemPartAlloc.status <> ERR_FUB_BUSY THEN

				IFmnTxt.Out.wSelectLanguageStatus := MNTXT_STAT_ERRMEM;
				_LoadState := _ls_error;

			END_IF

		_ls_load_instancetxt_03:

			_FileOpen(enable := TRUE, pDevice := ADR(KG_DEVICE_COMPACTFLASH), pFile := ADR('Language\Instance.csv'), mode := fiREAD_ONLY);

			IF _FileOpen.status = ERR_OK THEN

				_LoadState := _ls_load_instancetxt_04;

			ELSIF _FileOpen.status <> ERR_FUB_BUSY THEN

				IFmnTxt.Out.wSelectLanguageStatus := MNTXT_STAT_ERRINSTANCETXT;
				_LoadState := _ls_error;

			END_IF

		_ls_load_instancetxt_04:

			_FileRead(enable := TRUE, ident := _FileOpen.ident, offset := SIZEOF(KGBOM),pDest := _lAdrFile, len :=  _fiFileInfo.size-SIZEOF(KGBOM) );

			IF _FileRead.status <> ERR_FUB_BUSY THEN

				_LoadState := _ls_load_instancetxt_05;

			END_IF

		_ls_load_instancetxt_05:

			_FileClose(enable := TRUE, ident := _FileOpen.ident);

			IF _FileClose.status <> ERR_FUB_BUSY THEN

				IF _FileRead.status = ERR_OK THEN

					_LoadState := _ls_load_instancetxt_06;

				ELSE
					IFmnTxt.Out.wSelectLanguageStatus := MNTXT_STAT_ERRINSTANCETXT;
					_LoadState := _ls_error;

				END_IF

			END_IF

		_ls_load_instancetxt_06:

			// Zeilen in der Datei zählen und Startadressen ermitteln

			_CountLines.enable := TRUE;
			_CountLines.pFile := _lAdrFile;
			_CountLines.FileSize := _fiFileInfo.size - SIZEOF(KGBOM);
			_CountLines.MaxLines := MNTXT_MAXPARSELINES;
			_CountLines.pAdresses := _lAdrLineAdress;
			_CountLines.pLens := _lAdrLineLen;

			_CountLines();

			IF _CountLines.status = ERR_OK THEN

				_LoadState := _ls_load_instancetxt_07;

				_wStartLine := 1;
				_wIdxInstanceTxt := 0;
				_GetCsvDat.enable := TRUE;

			ELSE

				IFmnTxt.Out.wSelectLanguageStatus := MNTXT_STAT_ERRINSTANCETXT;
				_LoadState := _ls_error;

			END_IF

		_ls_load_instancetxt_07:

			// Datei parsen

			REPEAT

				brwcsncpy( ADR(_GetCsvDat.utfCsvString), _plLineAdress[_wStartLine], MIN(299, _pwLineLen[_wStartLine]));
				_GetCsvDat();
				_wStartLine := _wStartLine + 1;

				IF _GetCsvDat.RowType = 200 AND _GetCsvDat.csvTextRow.LCID = _wActLCID THEN

					_TxtLine.wNumber := _GetCsvDat.csvTextRow.TextNo;
					_TxtLine.wFunctionID := _GetCsvDat.csvTextRow.FunctionID;
					_TxtLine.utfText := _GetCsvDat.csvTextRow.utfText;

					_dowInstTxt(enable := TRUE, ident := _CheckDoInst.doId, Offset := SIZEOF(_TxtLine)*_wIdxInstanceTxt, pSource := ADR(_TxtLine), len := SIZEOF(_TxtLine));

					_wIdxInstanceTxt := _wIdxInstanceTxt + 1;

				END_IF

				_lCycleCounter := _lCycleCounter + 1;

				UNTIL

				_lCycleCounter > 20 OR _wIdxInstanceTxt > MNTXT_MAX_IDX_TXT_INSTANCE OR _wStartLine > _CountLines.CntLines

			END_REPEAT

			IF _wIdxInstanceTxt > MNTXT_MAX_IDX_TXT_INSTANCE OR _wStartLine > _CountLines.CntLines THEN

				IFmnTxt.Out.wCntInstanceTxt := _wIdxInstanceTxt;
				_LoadState := _ls_load_instancetxt_08;

			END_IF

		_ls_load_instancetxt_08:

			// Speicher frei geben

			_MemPartFree(enable := TRUE, ident := _MemPartCreate.ident, mem := _lAdrFile);

			IF _MemPartFree.status = ERR_OK THEN

				_LoadState := _ls_load_messagetxt_01;

			ELSIF _MemPartFree.status <> ERR_FUB_BUSY THEN

				IFmnTxt.Out.wSelectLanguageStatus := MNTXT_STAT_ERRINSTANCETXT;
				_LoadState := _ls_error;

			END_IF

		//###########################################################################################
		// MELDUNGSTEXTE LADEN
		//###########################################################################################

		_ls_load_messagetxt_01:

			// Nachsehen, ob Meldungstexte existieren

			IFmnTxt.Out.wCntMessageTxt := 0;
			IFmnTxt.Out.wCntMessageHlpTxt := 0;

			_FileInfo(enable := TRUE, pDevice := ADR(KG_DEVICE_COMPACTFLASH), pName := ADR('Messages\Messages.csv'), pInfo := ADR(_fiFileInfo));

			IF _FileInfo.status = ERR_OK THEN

				_LoadState := _ls_load_messagetxt_02;

			ELSIF _FileInfo.status <> ERR_FUB_BUSY THEN

				IFmnTxt.Out.wSelectLanguageStatus := MNTXT_STAT_ERRMESSAGETXT;
				_LoadState := _ls_error;

			END_IF

		_ls_load_messagetxt_02:

			// Speicher zum Parsen der Funktionstexte allokieren
			_MemPartAlloc(enable := TRUE, ident := _MemPartCreate.ident, len := _fiFileInfo.size-SIZEOF(KGBOM) );

			IF _MemPartAlloc.status = ERR_OK THEN

				_lAdrFile := _MemPartAlloc.mem;
				_LoadState := _ls_load_messagetxt_03;

			ELSIF _MemPartAlloc.status <> ERR_FUB_BUSY THEN

				IFmnTxt.Out.wSelectLanguageStatus := MNTXT_STAT_ERRMEM;
				_LoadState := _ls_error;

			END_IF

		_ls_load_messagetxt_03:

			_FileOpen(enable := TRUE, pDevice := ADR(KG_DEVICE_COMPACTFLASH), pFile := ADR('Messages\Messages.csv'), mode := fiREAD_ONLY);

			IF _FileOpen.status = ERR_OK THEN

				_LoadState := _ls_load_messagetxt_04;

			ELSIF _FileOpen.status <> ERR_FUB_BUSY THEN

				IFmnTxt.Out.wSelectLanguageStatus := MNTXT_STAT_ERRMESSAGETXT;
				_LoadState := _ls_error;

			END_IF

		_ls_load_messagetxt_04:

			_FileRead(enable := TRUE, ident := _FileOpen.ident, offset := SIZEOF(KGBOM),pDest := _lAdrFile, len :=  _fiFileInfo.size-SIZEOF(KGBOM) );

			IF _FileRead.status <> ERR_FUB_BUSY THEN

				_LoadState := _ls_load_messagetxt_05;

			END_IF

		_ls_load_messagetxt_05:

			_FileClose(enable := TRUE, ident := _FileOpen.ident);

			IF _FileClose.status <> ERR_FUB_BUSY THEN

				IF _FileRead.status = ERR_OK THEN

					_LoadState := _ls_load_messagetxt_06;

				ELSE
					IFmnTxt.Out.wSelectLanguageStatus := MNTXT_STAT_ERRMESSAGETXT;
					_LoadState := _ls_error;

				END_IF

			END_IF

		_ls_load_messagetxt_06:

			// Zeilen in der Datei zählen und Startadressen ermitteln

			_CountLines.enable := TRUE;
			_CountLines.pFile := _lAdrFile;
			_CountLines.FileSize := _fiFileInfo.size - SIZEOF(KGBOM);
			_CountLines.MaxLines := MNTXT_MAXPARSELINES;
			_CountLines.pAdresses := _lAdrLineAdress;
			_CountLines.pLens := _lAdrLineLen;

			_CountLines();

			IF _CountLines.status = ERR_OK THEN

				_LoadState := _ls_load_messagetxt_07;

				_wStartLine := 1;
				_wIdxMessageTxt := 0;
				_wIdxMessageHelpTxt := 0;
				_GetCsvDat.enable := TRUE;

			ELSE

				IFmnTxt.Out.wSelectLanguageStatus := MNTXT_STAT_ERRMESSAGETXT;
				_LoadState := _ls_error;

			END_IF

		_ls_load_messagetxt_07:

			// Datei parsen

			REPEAT

				brwcsncpy( ADR(_GetCsvDat.utfCsvString), _plLineAdress[_wStartLine], MIN(299, _pwLineLen[_wStartLine]));
				_GetCsvDat();
				_wStartLine := _wStartLine + 1;

				IF _GetCsvDat.RowType = 200 AND _GetCsvDat.csvTextRow.LCID = _wActLCID AND _wIdxMessageTxt < _lLenMsg THEN

					_TxtLine.wNumber := _GetCsvDat.csvTextRow.TextNo;
					_TxtLine.wFunctionID := _GetCsvDat.csvTextRow.FunctionID;
					_TxtLine.utfText := _GetCsvDat.csvTextRow.utfText;

					_dowMsgTxt(enable := TRUE, ident := _CheckDoMsg.doId, Offset := SIZEOF(_TxtLine)*_wIdxMessageTxt, pSource := ADR(_TxtLine), len := SIZEOF(_TxtLine));

					_wIdxMessageTxt := _wIdxMessageTxt + 1;

				ELSIF _GetCsvDat.RowType = 210 AND _GetCsvDat.csvHelpTextRow.LCID = _wActLCID AND _wIdxMessageHelpTxt < _lLenMsg THEN

					_TxtHelpLine.wNumber := _GetCsvDat.csvHelpTextRow.TextNo;
					_TxtHelpLine.wFunctionID := _GetCsvDat.csvHelpTextRow.FunctionID;
					_TxtHelpLine.utfText := _GetCsvDat.csvHelpTextRow.utfHelpText;

					_dowMsgHlpTxt(enable := TRUE, ident := _CheckDoMsgHlp.doId, Offset := SIZEOF(_TxtHelpLine)*_wIdxMessageHelpTxt, pSource := ADR(_TxtHelpLine), len := SIZEOF(_TxtHelpLine));

					_wIdxMessageHelpTxt := _wIdxMessageHelpTxt + 1;

				END_IF

				_lCycleCounter := _lCycleCounter + 1;

				UNTIL

				_lCycleCounter > 20 OR (_wIdxMessageTxt >= _lLenMsg AND _wIdxMessageHelpTxt >= _lLenMsg) OR _wStartLine > _CountLines.CntLines

			END_REPEAT

			IF (_wIdxMessageTxt >= _lLenMsg AND _wIdxMessageHelpTxt >= _lLenMsg) OR _wStartLine > _CountLines.CntLines THEN

				IFmnTxt.Out.wCntMessageTxt := _wIdxMessageTxt;
				IFmnTxt.Out.wCntMessageHlpTxt := _wIdxMessageHelpTxt;
				_LoadState := _ls_load_messagetxt_08;

			END_IF

		_ls_load_messagetxt_08:

			// Speicher frei geben

			_MemPartFree(enable := TRUE, ident := _MemPartCreate.ident, mem := _lAdrFile);

			IF _MemPartFree.status = ERR_OK THEN

				_LoadState := _ls_load_paramtxt_01;

			ELSIF _MemPartFree.status <> ERR_FUB_BUSY THEN

				IFmnTxt.Out.wSelectLanguageStatus := MNTXT_STAT_ERRMESSAGETXT;
				_LoadState := _ls_error;

			END_IF

		//###########################################################################################
		// PARAMETERTEXTE LADEN
		//###########################################################################################

		_ls_load_paramtxt_01:

			// Nachsehen, ob Parametertexte existieren

			IFmnTxt.Out.wCntParamTxt := 0;
			IFmnTxt.Out.wCntParamHlpTxt := 0;

			IF MNTXT_LOAD_PARAMETERTEXT AND _CheckDoPar.doId <> 0 THEN

				_FileInfo(enable := TRUE, pDevice := ADR(KG_DEVICE_COMPACTFLASH), pName := ADR('Language\ParamTxt.csv'), pInfo := ADR(_fiFileInfo));

				IF _FileInfo.status = ERR_OK THEN

					_LoadState := _ls_load_paramtxt_02;

				ELSIF _FileInfo.status <> ERR_FUB_BUSY THEN

					IFmnTxt.Out.wSelectLanguageStatus := MNTXT_STAT_ERRPARAMTXT;
					_LoadState := _ls_error;

				END_IF

			ELSE

				_LoadState := _ls_idle;
				IFmnTxt.Out.wSelectLanguageStatus := MNTXT_STAT_OK;

			END_IF

		_ls_load_paramtxt_02:

			// Speicher zum Parsen der Parametertexte allokieren
			_MemPartAlloc(enable := TRUE, ident := _MemPartCreate.ident, len := _fiFileInfo.size-SIZEOF(KGBOM) );

			IF _MemPartAlloc.status = ERR_OK THEN

				_lAdrFile := _MemPartAlloc.mem;
				_LoadState := _ls_load_paramtxt_03;

			ELSIF _MemPartAlloc.status <> ERR_FUB_BUSY THEN

				IFmnTxt.Out.wSelectLanguageStatus := MNTXT_STAT_ERRMEM;
				_LoadState := _ls_error;

			END_IF

		_ls_load_paramtxt_03:

			_FileOpen(enable := TRUE, pDevice := ADR(KG_DEVICE_COMPACTFLASH), pFile := ADR('Language\ParamTxt.csv'), mode := fiREAD_ONLY);

			IF _FileOpen.status = ERR_OK THEN

				_LoadState := _ls_load_paramtxt_04;

			ELSIF _FileOpen.status <> ERR_FUB_BUSY THEN

				IFmnTxt.Out.wSelectLanguageStatus := MNTXT_STAT_ERRPARAMTXT;
				_LoadState := _ls_error;

			END_IF

		_ls_load_paramtxt_04:

			_FileRead(enable := TRUE, ident := _FileOpen.ident, offset := SIZEOF(KGBOM),pDest := _lAdrFile, len :=  _fiFileInfo.size-SIZEOF(KGBOM) );

			IF _FileRead.status <> ERR_FUB_BUSY THEN

				_LoadState := _ls_load_paramtxt_05;

			END_IF

		_ls_load_paramtxt_05:

			_FileClose(enable := TRUE, ident := _FileOpen.ident);

			IF _FileClose.status <> ERR_FUB_BUSY THEN

				IF _FileRead.status = ERR_OK THEN

					_LoadState := _ls_load_paramtxt_06;

				ELSE
					IFmnTxt.Out.wSelectLanguageStatus := MNTXT_STAT_ERRPARAMTXT;
					_LoadState := _ls_error;

				END_IF

			END_IF

		_ls_load_paramtxt_06:

			// Zeilen in der Datei zählen und Startadressen ermitteln

			_CountLines.enable := TRUE;
			_CountLines.pFile := _lAdrFile;
			_CountLines.FileSize := _fiFileInfo.size - SIZEOF(KGBOM);
			_CountLines.MaxLines := MNTXT_MAXPARSELINES;
			_CountLines.pAdresses := _lAdrLineAdress;
			_CountLines.pLens := _lAdrLineLen;

			_CountLines();

			IF _CountLines.status = ERR_OK THEN

				_LoadState := _ls_load_paramtxt_07;

				_wStartLine := 1;
				_wIdxParamTxt := 0;
				_wIdxParamHelpTxt := 0;
				_GetCsvDat.enable := TRUE;

			ELSE

				IFmnTxt.Out.wSelectLanguageStatus := MNTXT_STAT_ERRPARAMTXT;
				_LoadState := _ls_error;

			END_IF

		_ls_load_paramtxt_07:

			// Datei parsen

			REPEAT

				brwcsncpy( ADR(_GetCsvDat.utfCsvString), _plLineAdress[_wStartLine], MIN(299, _pwLineLen[_wStartLine]));
				_GetCsvDat();
				_wStartLine := _wStartLine + 1;

				IF _GetCsvDat.RowType = 200 AND _GetCsvDat.csvTextRow.LCID = _wActLCID AND _wIdxParamTxt <= MNTXT_MAX_IDX_TXT_PARAMETER THEN

					_TxtLine.wNumber := _GetCsvDat.csvTextRow.TextNo;
					_TxtLine.wFunctionID := _GetCsvDat.csvTextRow.FunctionID;
					_TxtLine.utfText := _GetCsvDat.csvTextRow.utfText;

					_dowParTxt(enable := TRUE, ident := _CheckDoPar.doId, Offset := SIZEOF(_TxtLine)*_wIdxParamTxt, pSource := ADR(_TxtLine), len := SIZEOF(_TxtLine));

					_wIdxParamTxt := _wIdxParamTxt + 1;

				ELSIF _GetCsvDat.RowType = 210 AND _GetCsvDat.csvHelpTextRow.LCID = _wActLCID AND _wIdxParamHelpTxt <= MNTXT_MAX_IDX_TXT_PARAMETER AND MNTXT_LOAD_PARAMTERHELPTEXT THEN

					_TxtHelpLine.wNumber := _GetCsvDat.csvHelpTextRow.TextNo;
					_TxtHelpLine.wFunctionID := _GetCsvDat.csvHelpTextRow.FunctionID;
					_TxtHelpLine.utfText := _GetCsvDat.csvHelpTextRow.utfHelpText;

					_dowParHlpTxt(enable := TRUE, ident := _CheckDoParHlp.doId, Offset := SIZEOF(_TxtHelpLine)*_wIdxParamHelpTxt, pSource := ADR(_TxtHelpLine), len := SIZEOF(_TxtHelpLine));

					_wIdxParamHelpTxt := _wIdxParamHelpTxt + 1;

				END_IF

				_lCycleCounter := _lCycleCounter + 1;

				UNTIL

				_lCycleCounter > 20 OR (_wIdxParamTxt > MNTXT_MAX_IDX_TXT_PARAMETER AND _wIdxParamHelpTxt > MNTXT_MAX_IDX_TXT_PARAMETER) OR _wStartLine > _CountLines.CntLines

			END_REPEAT

			IF (_wIdxParamTxt > MNTXT_MAX_IDX_TXT_PARAMETER AND _wIdxParamHelpTxt > MNTXT_MAX_IDX_TXT_PARAMETER) OR _wStartLine > _CountLines.CntLines THEN

				IFmnTxt.Out.wCntParamTxt := _wIdxParamTxt;
				IFmnTxt.Out.wCntParamHlpTxt := _wIdxParamHelpTxt;
				_LoadState := _ls_load_paramtxt_08;

			END_IF

		_ls_load_paramtxt_08:

			// Speicher frei geben

			_MemPartFree(enable := TRUE, ident := _MemPartCreate.ident, mem := _lAdrFile);

			IF _MemPartFree.status = ERR_OK THEN

				_LoadState := _ls_idle;
				IFmnTxt.Out.wSelectLanguageStatus := MNTXT_STAT_OK;

			ELSIF _MemPartFree.status <> ERR_FUB_BUSY THEN

				IFmnTxt.Out.wSelectLanguageStatus := MNTXT_STAT_ERRPARAMTXT;
				_LoadState := _ls_error;

			END_IF

		_ls_error:

			// Fehlerzustand

	END_CASE

END_PROGRAM
```

#### mnTxtInit.st - Initialization code
```iecst
(********************************************************************
 * COPYRIGHT -- Herbert Kannegiesser GmbH
 ********************************************************************
 * Program: mnTxt
 * File: mnTxtInit.st
 * Author: hunholz
 * Created: November 25, 2011
 ********************************************************************
 * Implementation of program mnTxt
 ********************************************************************)

PROGRAM _INIT

	// Packet-Version auslesen mit MO_ver aus SYS_lib und für den Additional Status zur Verfügung stellen

	_sPkgName := 'mnTxt';

	IF ( MO_ver(ADR(_sPkgName), 0, ADR(_VerStruc)) = 0 ) THEN

		brsmemcpy(ADR(mnTxtStatAd.sPkgVersion), ADR(_VerStruc.version), SIZEOF(_VerStruc.version));

	ELSE

		mnTxtStatAd.sPkgVersion := '---';

	END_IF

	brsmemset(ADR(IFmnTxt.Out), 0, SIZEOF(IFmnTxt.Out));

	IFmnTxt.Out.wSelectLanguageStatus := MNTXT_STAT_INIT;

	REPEAT

		//===================================
		// Speicher zum Parsen bereitstellen
		//===================================

		// Bedarf berechnen

		_lLineMem := (((SIZEOF(_plLineAdress) + SIZEOF(_pwLineLen)) / 8) + 2 ) * 8;

		_lLineMem := _lLineMem + ((MNTXT_TEMPREADCSVSIZE / 8) + 2) * 8;

		_lLineMem := _lLineMem + 1000;

		_MemPartCreate(enable := TRUE, len := _lLineMem);

		IF _MemPartCreate.status <> ERR_OK THEN

			IFmnTxt.Out.wSelectLanguageStatus := MNTXT_STAT_ERRMEM;
			EXIT;

		END_IF

		// Zeilenadresstabelle
		_MemPartAlloc(enable := TRUE, ident := _MemPartCreate.ident, len := SIZEOF(_plLineAdress) + SIZEOF(_pwLineLen) );

		IF _MemPartAlloc.status <> ERR_OK THEN

			IFmnTxt.Out.wSelectLanguageStatus := MNTXT_STAT_ERRMEM;
			EXIT;

		END_IF

		_lAdrLineAdress := _MemPartAlloc.mem;
		_plLineAdress ACCESS _lAdrLineAdress;

		_lAdrLineLen := _lAdrLineAdress + SIZEOF(_plLineAdress);
		_pwLineLen ACCESS _lAdrLineLen;

		//LCID_Tabelle einlesen

		_FileInfo(enable := TRUE, pDevice := ADR(KG_DEVICE_COMPACTFLASH), pName := ADR('Language\lcid.csv'), pInfo := ADR(_fiFileInfo));

		IF _FileInfo.status <> ERR_OK THEN

			IFmnTxt.Out.wSelectLanguageStatus := MNTXT_STAT_ERRLCID;
			EXIT;

		END_IF

		_MemPartAlloc(enable := TRUE, ident := _MemPartCreate.ident, len := _fiFileInfo.size-SIZEOF(KGBOM) );

		IF _MemPartAlloc.status <> ERR_OK THEN

			IFmnTxt.Out.wSelectLanguageStatus := MNTXT_STAT_ERRMEM;
			EXIT;

		END_IF

		_lAdrFile := _MemPartAlloc.mem;

		_FileOpen(enable := TRUE, pDevice := ADR(KG_DEVICE_COMPACTFLASH), pFile := ADR('Language\lcid.csv'), mode := fiREAD_ONLY);

		IF _FileOpen.status <> ERR_OK THEN

			IFmnTxt.Out.wSelectLanguageStatus := MNTXT_STAT_ERRLCID;
			EXIT;

		END_IF

		_FileRead(enable := TRUE, ident := _FileOpen.ident, offset := SIZEOF(KGBOM),pDest := _lAdrFile, len :=  _fiFileInfo.size-SIZEOF(KGBOM) ) ;

		_FileClose(enable := TRUE, ident := _FileOpen.ident);

		IF _FileRead.status <> ERR_OK THEN

			IFmnTxt.Out.wSelectLanguageStatus := MNTXT_STAT_ERRLCID;
			EXIT;

		END_IF

		// Zeilen in der Datei zählen und Startadressen ermitteln

		_CountLines.enable := TRUE;
		_CountLines.pFile := _lAdrFile;
		_CountLines.FileSize := _fiFileInfo.size - SIZEOF(KGBOM);
		_CountLines.MaxLines := MNTXT_MAXPARSELINES;
		_CountLines.pAdresses := _lAdrLineAdress;
		_CountLines.pLens := _lAdrLineLen;

		_CountLines();

		IF _CountLines.status <> ERR_OK THEN

			IFmnTxt.Out.wSelectLanguageStatus := MNTXT_STAT_ERRLCID;
			EXIT;

		END_IF

		// Zeilen auslesen und LCID-Werte ermitteln

		_xGermanExist := FALSE;
		_wStartLine := 1;
		_wIdxLCID := 0;
		_GetCsvDat.enable := TRUE;

		REPEAT

			brwcsncpy( ADR(_GetCsvDat.utfCsvString), _plLineAdress[_wStartLine], MIN(299, _pwLineLen[_wStartLine]));
			_GetCsvDat();
			_wStartLine := _wStartLine + 1;

			IF _GetCsvDat.RowType = 248 AND _GetCsvDat.CsvLCIDrow.LCID > 0 THEN

				IFmnTxt.Out.wLCIDs[_wIdxLCID] := _GetCsvDat.CsvLCIDrow.LCID;
				_wIdxLCID := _wIdxLCID + 1;

				IF _GetCsvDat.CsvLCIDrow.LCID = MNTXT_LCID_GERMAN THEN
					_xGermanExist := TRUE;
				END_IF

			END_IF

			UNTIL
			_wIdxLCID > MNTXT_MAX_IDX_LCID OR _wStartLine > _CountLines.CntLines
		END_REPEAT

		IFmnTxt.Out.wCntLCID := _wIdxLCID;

		_MemPartFree(enable := TRUE, ident := _MemPartCreate.ident, mem := _lAdrFile);

		IF IFmnTxt.Out.wCntLCID = 0 THEN

			IFmnTxt.Out.wSelectLanguageStatus := MNTXT_STAT_ERRLCID;
			EXIT;

		END_IF

		//##############################################################################

		IFmnTxt.Out.wSelectLanguageStatus := MNTXT_STAT_NOLANGUAGE;

		_initState := _is_checkFunctionTxt;
		_xInitOK := FALSE;
		_xInitDone := FALSE;

		UNTIL
		TRUE
	END_REPEAT

	REPEAT

		CASE _initState OF

			// Datenobjekte für Funktionstexte prüfen und ggf. anlegen
			_is_checkFunctionTxt:

				IFmnTxt.Out.ptrFunctionTxtList := 0;
				IFmnTxt.Out.wCntFunctionTxt := 0;

				_lLenFuncTxt := SIZEOF(_TxtLine)*(MNTXT_MAX_IDX_TXT_FUNCTION+1);

				IF MNTXT_LOAD_FUNCTIONTEXT THEN

					_CheckDoFunc(Enable := TRUE, pName := ADR(MNTXT_DATOBJNAME_FUNTXT), MinLen := _lLenFuncTxt, NomLen := _lLenFuncTxt, Create := TRUE, MemType := doUSRROM);

					IF _CheckDoFunc.Status <> ERR_FUB_BUSY THEN

						// DO mit Templatetexten füllen, wenn es neu angelegt wurde

						IF _CheckDoFunc.Status = KG_INFO_DO_NEW OR _CheckDoFunc.Status = ERR_OK THEN

							_debFunctionTxtList ACCESS _CheckDoFunc.doMem;

							IFmnTxt.Out.ptrFunctionTxtList := _CheckDoFunc.doMem;

							IF _CheckDoFunc.Status = KG_INFO_DO_NEW THEN

								_initState := _is_writeFunctionTxt;
								_ii := 0;

							ELSE

								_initState := _is_checkInstanceTxt;

							END_IF

						ELSE

							_xInitDone := TRUE;
							IFmnTxt.Out.wSelectLanguageStatus := _CheckDoFunc.Status;

						END_IF

					END_IF

				ELSE

					_initState := _is_checkInstanceTxt;

				END_IF

			_is_writeFunctionTxt:

				REPEAT

					_TxtLine.wNumber 		:= _ii;
					_TxtLine.wFunctionID 	:= _ii;
					_TxtLine.utfText		:= "Function";
					_utfNo					:= UINT_TO_WSTRING(_ii);
					brwcscat(ADR(_TxtLine.utfText), ADR(_utfNo));

					_dowFuncTxt(enable := TRUE, ident := _CheckDoFunc.doId, Offset := SIZEOF(_TxtLine)*_ii, pSource := ADR(_TxtLine), len := SIZEOF(_TxtLine));

					IF _dowFuncTxt.status <> ERR_OK THEN

						IFmnTxt.Out.wSelectLanguageStatus := MNTXT_STAT_ERRDATOBJ;
						_xInitDone := TRUE;
						EXIT;

					END_IF

					_ii := _ii + 1;

					UNTIL
					((_ii MOD 10) = 0) OR _ii > MNTXT_MAX_IDX_TXT_FUNCTION
				END_REPEAT

				IF _ii > MNTXT_MAX_IDX_TXT_FUNCTION THEN

					_initState := _is_checkInstanceTxt;

				END_IF

			// Datenobjekte für Instanztexte prüfen und ggf. anlegen
			_is_checkInstanceTxt:

				IFmnTxt.Out.ptrInstanceTxtList := 0;
				IFmnTxt.Out.wCntInstanceTxt		:= 0;

				_lLenInstTxt := SIZEOF(_TxtLine)*(MNTXT_MAX_IDX_TXT_INSTANCE + 1);

				IF MNTXT_LOAD_INSTANCETEXT THEN

					_CheckDoInst(Enable := TRUE, pName := ADR(MNTXT_DATOBJNAME_INSTXT), MinLen := _lLenInstTxt, NomLen := _lLenInstTxt, Create := TRUE, MemType := doUSRROM);

					IF _CheckDoInst.Status <> ERR_FUB_BUSY THEN

						// DO mit Templatetexten füllen, wenn es neu angelegt wurde

						IF _CheckDoInst.Status = KG_INFO_DO_NEW OR _CheckDoInst.Status = ERR_OK THEN

							IFmnTxt.Out.ptrInstanceTxtList := _CheckDoInst.doMem;

							_debInstanceTxtList ACCESS _CheckDoInst.doMem;

							IF _CheckDoInst.Status = KG_INFO_DO_NEW THEN

								_ii := 0;
								_initState := _is_writeInstanceTxt;

							ELSE

								_initState := _is_checkParTxt;

							END_IF

						ELSE

							IFmnTxt.Out.wSelectLanguageStatus := _CheckDoInst.Status;
							_xInitDone := TRUE;

						END_IF

					END_IF

				ELSE

					_initState := _is_checkParTxt;

				END_IF

			_is_writeInstanceTxt:

				REPEAT

					_TxtLine.wNumber 		:= _ii;
					_TxtLine.wFunctionID 	:= _ii;
					_TxtLine.utfText		:= "Instance";
					_utfNo					:= UINT_TO_WSTRING(_ii);
					brwcscat(ADR(_TxtLine.utfText), ADR(_utfNo));

					_dowInstTxt(enable := TRUE, ident := _CheckDoInst.doId, Offset := SIZEOF(_TxtLine)*_ii, pSource := ADR(_TxtLine), len := SIZEOF(_TxtLine));

					IF _dowInstTxt.status <> ERR_OK THEN

						IFmnTxt.Out.wSelectLanguageStatus := MNTXT_STAT_ERRDATOBJ;
						_xInitDone := TRUE;
						EXIT;

					END_IF

					_ii := _ii + 1;

					UNTIL
					((_ii MOD 10) = 0) OR _ii > MNTXT_MAX_IDX_TXT_INSTANCE
				END_REPEAT

				IF _ii > MNTXT_MAX_IDX_TXT_INSTANCE THEN

					_initState := _is_checkParTxt;

				END_IF

			// Datenobjekte für Parametertexte prüfen und ggf. anlegen
			_is_checkParTxt:

				IFmnTxt.Out.ptrParamTxtList := 0;
				IFmnTxt.Out.wCntParamTxt := 0;

				_lLenParTxt := SIZEOF(_TxtLine)*(MNTXT_MAX_IDX_TXT_PARAMETER + 1);

				IF MNTXT_LOAD_PARAMETERTEXT THEN

					_CheckDoPar(Enable := TRUE, pName := ADR(MNTXT_DATOBJNAME_PARTXT), MinLen := _lLenParTxt, NomLen := _lLenParTxt, Create := TRUE, MemType := doUSRROM);

					IF _CheckDoPar.Status <> ERR_FUB_BUSY THEN

						// DO mit Templatetexten füllen, wenn es neu angelegt wurde

						IF _CheckDoPar.Status = KG_INFO_DO_NEW OR _CheckDoPar.Status = ERR_OK THEN

							_debParameterTxtList ACCESS _CheckDoPar.doMem;

							IFmnTxt.Out.ptrParamTxtList := _CheckDoPar.doMem;

							IF _CheckDoPar.Status = KG_INFO_DO_NEW THEN

								_ii := 0;
								_initState := _is_writeParTxt;

							ELSE

								_initState := _is_checkParHlpTxt;

							END_IF

						ELSE

							IFmnTxt.Out.wSelectLanguageStatus := _CheckDoPar.Status;
							_xInitDone := TRUE;

						END_IF

					END_IF

				ELSE

					_initState := _is_checkParHlpTxt;

				END_IF

			_is_writeParTxt:

				REPEAT

					_TxtLine.wNumber 		:= _ii;
					_TxtLine.wFunctionID 	:= _ii;
					_TxtLine.utfText		:= "Parameter";
					_utfNo					:= UINT_TO_WSTRING(_ii);
					brwcscat(ADR(_TxtLine.utfText), ADR(_utfNo));

					_dowParTxt(enable := TRUE, ident := _CheckDoPar.doId, Offset := SIZEOF(_TxtLine)*_ii, pSource := ADR(_TxtLine), len := SIZEOF(_TxtLine));

					IF _dowParTxt.status <> ERR_OK THEN

						IFmnTxt.Out.wSelectLanguageStatus := MNTXT_STAT_ERRDATOBJ;
						_xInitDone := TRUE;
						EXIT;

					END_IF

					_ii := _ii + 1;

					UNTIL
					((_ii MOD 10) = 0) OR _ii > MNTXT_MAX_IDX_TXT_PARAMETER
				END_REPEAT

				IF _ii > MNTXT_MAX_IDX_TXT_PARAMETER THEN

					_initState := _is_checkParHlpTxt;

				END_IF

			// Datenobjekte für Parameterhilfstexte prüfen und ggf. anlegen
			_is_checkParHlpTxt:

				IFmnTxt.Out.ptrParamHelpTxtList := 0;
				IFmnTxt.Out.wCntParamHlpTxt := 0;

				_lLenParHlpTxt := SIZEOF(_TxtHelpLine)*(MNTXT_MAX_IDX_TXT_PARAMETER + 1);

				IF MNTXT_LOAD_PARAMTERHELPTEXT THEN

					_CheckDoParHlp(Enable := TRUE, pName := ADR(MNTXT_DATOBJNAME_PARHELPTXT), MinLen := _lLenParHlpTxt, NomLen := _lLenParHlpTxt, Create := TRUE, MemType := doUSRROM);

					IF _CheckDoParHlp.Status <> ERR_FUB_BUSY THEN

						// DO mit Templatetexten füllen, wenn es neu angelegt wurde

						IF _CheckDoParHlp.Status = KG_INFO_DO_NEW OR _CheckDoParHlp.Status = ERR_OK THEN

							_debParameterHlpTxtList ACCESS _CheckDoParHlp.doMem;

							IFmnTxt.Out.ptrParamHelpTxtList := _CheckDoParHlp.doMem;

							IF _CheckDoParHlp.Status = KG_INFO_DO_NEW THEN

								_ii := 0;
								_initState := _is_writeParHlpTxt;

							ELSE

								_initState := _is_checkMsgCnt;

							END_IF

						ELSE

							IFmnTxt.Out.wSelectLanguageStatus := _CheckDoParHlp.Status;
							_xInitDone := TRUE;

						END_IF

					END_IF

				ELSE

					_initState := _is_checkMsgCnt;

				END_IF

			_is_writeParHlpTxt:

				REPEAT

					_TxtHelpLine.wNumber 		:= _ii;
					_TxtHelpLine.wFunctionID 	:= _ii;
					_TxtHelpLine.utfText		:= "Parameter Help";
					_utfNo						:= UINT_TO_WSTRING(_ii);
					brwcscat(ADR(_TxtHelpLine.utfText), ADR(_utfNo));

					_dowParHlpTxt(enable := TRUE, ident := _CheckDoParHlp.doId, Offset := SIZEOF(_TxtHelpLine)*_ii, pSource := ADR(_TxtHelpLine), len := SIZEOF(_TxtHelpLine));

					IF _dowParHlpTxt.status <> ERR_OK THEN

						IFmnTxt.Out.wSelectLanguageStatus := MNTXT_STAT_ERRDATOBJ;
						_xInitDone := TRUE;
						EXIT;

					END_IF

					_ii := _ii + 1;

					UNTIL
					((_ii MOD 10) =0) OR _ii > MNTXT_MAX_IDX_TXT_PARAMETER
				END_REPEAT

				IF _ii > MNTXT_MAX_IDX_TXT_PARAMETER THEN

					_initState := _is_checkMsgCnt;

				END_IF

			// Anzahl Meldungen ermitteln
			_is_checkMsgCnt:

				REPEAT

					_doiMsgCfg(enable := TRUE, pName := ADR('CfgMsgStat'));

					IF _doiMsgCfg.status <> ERR_OK THEN

						IFmnTxt.Out.wSelectLanguageStatus := MNTXT_STAT_ERRMSGCFG;
						_xInitDone := TRUE;
						EXIT;

					END_IF

					IF _doiMsgCfg.len < 2 THEN

						IFmnTxt.Out.wSelectLanguageStatus := MNTXT_STAT_ERRMSGCFG;
						_xInitDone := TRUE;
						EXIT;

					END_IF

					_MsgCfgList ACCESS _doiMsgCfg.pDatObjMem + 2;

					_lLenMsg := (_doiMsgCfg.len-2) / SIZEOF(_MsgCfgList[0]);

					_initState := _is_checkMsgTxt;

					UNTIL
					TRUE

				END_REPEAT

			// Datenobjekte für Meldungstexte prüfen und ggf. anlegen
			_is_checkMsgTxt:

				// Referenz auf die Meldungskonfiguration holen und Anzahl der möglichen Meldungen
				// ermitteln

				IFmnTxt.Out.ptrMessageTxtList := 0;
				IFmnTxt.Out.wCntMessageTxt := 0;

				_lLenMsgTxt := SIZEOF(_TxtLine)* _lLenMsg;

				_CheckDoMsg(Enable := TRUE, pName := ADR(MNTXT_DATOBJNAME_MSGTXT), MinLen := _lLenMsgTxt, NomLen := _lLenMsgTxt, Create := TRUE, MemType := doUSRROM);

				IF _CheckDoMsg.Status <> ERR_FUB_BUSY THEN

					// DO mit Templatetexten füllen, wenn es neu angelegt wurde
					IF _CheckDoMsg.Status = KG_INFO_DO_NEW OR _CheckDoMsg.Status = ERR_OK THEN

						_debMessageTxtList ACCESS _CheckDoMsg.doMem;

						IFmnTxt.Out.ptrMessageTxtList := _CheckDoMsg.doMem;
						IFmnTxt.Out.wCntMessageTxt := UDINT_TO_UINT(_lLenMsg);

						_ii := 0;

						_initState := _is_writeMsgTxt;

					ELSE

						IFmnTxt.Out.wSelectLanguageStatus := _CheckDoMsg.Status;
						_xInitDone := TRUE;

					END_IF

				END_IF

			_is_writeMsgTxt:

				IF _CheckDoMsg.Status = KG_INFO_DO_NEW AND _lLenMsg > 0 THEN

					REPEAT

						_TxtLine.wNumber 		:= _MsgCfgList[_ii].wMsgNumber;
						_TxtLine.wFunctionID 	:= _MsgCfgList[_ii].wFunction_ID;
						_TxtLine.wInstance		:= _MsgCfgList[_ii].wInstance;
						_TxtLine.utfText		:= "Message";
						_utfNo					:= UINT_TO_WSTRING(_MsgCfgList[_ii].wMsgNumber);
						brwcscat(ADR(_TxtLine.utfText), ADR(_utfNo));

						_dowMsgTxt(enable := TRUE, ident := _CheckDoMsg.doId, Offset := SIZEOF(_TxtLine)*_ii, pSource := ADR(_TxtLine), len := SIZEOF(_TxtLine));

						IF _dowMsgTxt.status <> ERR_OK THEN

							IFmnTxt.Out.wSelectLanguageStatus := MNTXT_STAT_ERRDATOBJ;
							_xInitDone := TRUE;
							EXIT;

						END_IF

						_ii := _ii + 1;

						UNTIL
						((_ii MOD 10) = 0) OR _ii >= _lLenMsg

					END_REPEAT

					IF _ii >= _lLenMsg THEN

						_initState := _is_checkMsgHlpTxt;

					END_IF

				ELSE

					_initState := _is_checkMsgHlpTxt;

				END_IF

			// Datenobjekte für Meldungstexte prüfen und ggf. anlegen
			_is_checkMsgHlpTxt:

				IFmnTxt.Out.ptrMessageHelpTxtList := 0;
				IFmnTxt.Out.wCntMessageHlpTxt := 0;

				_lLenMsgHlpTxt := SIZEOF(_TxtHelpLine)* _lLenMsg;

				_CheckDoMsgHlp(Enable := TRUE, pName := ADR(MNTXT_DATOBJNAME_MSGHELPTXT), MinLen := _lLenMsgHlpTxt, NomLen := _lLenMsgHlpTxt, Create := TRUE, MemType := doUSRROM);

				IF _CheckDoMsgHlp.Status <> ERR_FUB_BUSY THEN

					// DO mit Templatetexten füllen, wenn es neu angelegt wurde
					IF _CheckDoMsgHlp.Status = KG_INFO_DO_NEW OR _CheckDoMsgHlp.Status = ERR_OK THEN

						_debMessageHlpTxtList ACCESS _CheckDoMsgHlp.doMem;

						IFmnTxt.Out.ptrMessageHelpTxtList := _CheckDoMsgHlp.doMem;
						IFmnTxt.Out.wCntMessageHlpTxt := UDINT_TO_UINT(_lLenMsg);

						_ii := 0;

						_initState := _is_writeMsgHlpTxt;

					ELSE

						IFmnTxt.Out.wSelectLanguageStatus := _CheckDoMsg.Status;
						_xInitDone := TRUE;

					END_IF

				END_IF

			_is_writeMsgHlpTxt:

				IF _CheckDoMsgHlp.Status = KG_INFO_DO_NEW AND _lLenMsg > 0 THEN

					REPEAT

						_TxtHelpLine.wNumber 		:= _MsgCfgList[_ii].wMsgNumber;
						_TxtHelpLine.wFunctionID 	:= _MsgCfgList[_ii].wFunction_ID;
						_TxtHelpLine.wInstance		:= _MsgCfgList[_ii].wInstance;
						_TxtHelpLine.utfText		:= "Message Help";
						_utfNo					:= UINT_TO_WSTRING(_MsgCfgList[_ii].wMsgNumber);
						brwcscat(ADR(_TxtHelpLine.utfText), ADR(_utfNo));

						_dowMsgHlpTxt(enable := TRUE, ident := _CheckDoMsgHlp.doId, Offset := SIZEOF(_TxtHelpLine)*_ii, pSource := ADR(_TxtHelpLine), len := SIZEOF(_TxtHelpLine));

						IF _dowMsgHlpTxt.status <> ERR_OK THEN

							IFmnTxt.Out.wSelectLanguageStatus := MNTXT_STAT_ERRDATOBJ;
							_xInitDone := TRUE;
							EXIT;

						END_IF

						_ii := _ii + 1;

						UNTIL
						((_ii MOD 10)) = 0 OR	_ii >= _lLenMsg
					END_REPEAT

					IF _ii >= _lLenMsg THEN
						_xInitDone := TRUE;
						_xInitOK := TRUE;
					END_IF

				ELSE

					_xInitDone := TRUE;
					_xInitOK := TRUE;

				END_IF

		END_CASE

		UNTIL
		_xInitDone
	END_REPEAT

END_PROGRAM
```

#### mnTxt.var - Local variables
```iecst
(********************************************************************
 * COPYRIGHT -- Herbert Kannegiesser GmbH
 ********************************************************************
 * Program: mnTxt
 * File: mnTxt.var
 * Author: hunholz
 * Created: November 25, 2011
 ********************************************************************
 * Local variables of program mnTxt
 ********************************************************************)
(*Hilfsvariablen*)
VAR
	_ii : UINT;
	_utfNo : WSTRING[5];
	_TxtLine : mnTxt_TxtLine_Typ;
	_TxtHelpLine : mnTxt_HelpTxtLine_Typ;
END_VAR
(*Function-Txt Datenobjekt prüfen, anlegen, füllen*)
VAR
	_dowFuncTxt : DatObjWrite;
	_debFunctionTxtList : REFERENCE TO ARRAY[0..MNTXT_MAX_IDX_TXT_FUNCTION] OF mnTxt_TxtLine_Typ;
	_lLenFuncTxt : UDINT;
END_VAR
(*Instance-Txt Datenobjekt prüfen, anlegen, füllen*)
VAR
	_dowInstTxt : DatObjWrite;
	_debInstanceTxtList : REFERENCE TO ARRAY[0..MNTXT_MAX_IDX_TXT_INSTANCE] OF mnTxt_TxtLine_Typ;
	_lLenInstTxt : UDINT;
END_VAR
(*Parameter-Txt Datenobjekt prüfen, anlegen, füllen*)
VAR
	_dowParTxt : DatObjWrite;
	_debParameterTxtList : REFERENCE TO ARRAY[0..MNTXT_MAX_IDX_TXT_PARAMETER] OF mnTxt_TxtLine_Typ;
	_lLenParTxt : UDINT;
END_VAR
(*Parameter-HlpTxt Datenobjekt prüfen, anlegen, füllen*)
VAR
	_dowParHlpTxt : DatObjWrite;
	_debParameterHlpTxtList : REFERENCE TO ARRAY[0..MNTXT_MAX_IDX_TXT_PARAMETER] OF mnTxt_HelpTxtLine_Typ;
	_lLenParHlpTxt : UDINT;
END_VAR
(*Meldungs-Txt Datenobjekt prüfen, anlegen, füllen*)
VAR
	_dowMsgTxt : DatObjWrite;
	_debMessageTxtList : REFERENCE TO ARRAY[0..65535] OF mnTxt_TxtLine_Typ;
	_lLenMsgTxt : UDINT;
END_VAR
(*Meldungs-HlpTxt Datenobjekt prüfen, anlegen, füllen*)
VAR
	_dowMsgHlpTxt : DatObjWrite;
	_debMessageHlpTxtList : REFERENCE TO ARRAY[0..65535] OF mnTxt_HelpTxtLine_Typ;
	_lLenMsgHlpTxt : UDINT;
	_doiMsgCfg : DatObjInfo;
	_lLenMsg : UDINT;
	_MsgCfgList : REFERENCE TO ARRAY[0..65535] OF MsgCfgLine_Typ;
	_LoadState : _mntxt_loadstate_enum;
END_VAR
VAR CONSTANT
	_MemPartCreate : AsMemPartCreate := (0);
END_VAR
VAR
	_MemPartAlloc : AsMemPartAlloc;
	_plLineAdress : REFERENCE TO ARRAY[1..MNTXT_MAXPARSELINES] OF UDINT;
	_pwLineLen : REFERENCE TO ARRAY[1..MNTXT_MAXPARSELINES] OF UINT;
	_fiFileInfo : fiFILE_INFO;
	_FileInfo : FileInfo;
	_FileOpen : FileOpen;
	_lAdrFile : UDINT;
	_FileRead : FileRead;
	_FileClose : FileClose;
	_CountLines : mnParam_CountLines;
	_lAdrLineAdress : UDINT;
	_lAdrLineLen : UDINT;
	_wStartLine : UINT;
	_wIdxLCID : UINT;
	_GetCsvDat : mnParam_GetCsvDat;
	_MemPartFree : AsMemPartFree;
END_VAR
VAR RETAIN
	_wActLCID : UINT;
END_VAR
VAR
	_xGermanExist : BOOL;
	_lCycleCounter : UDINT;
	_wIdxFunctionTxt : UINT;
	_wIdxInstanceTxt : UINT;
	_wIdxMessageTxt : UINT;
	_wIdxMessageHelpTxt : UINT;
	_wIdxParamTxt : UINT;
	_wIdxParamHelpTxt : UINT;
	_sPkgName : STRING[11];
	_VerStruc : MoVerStruc_typ;
	_lLineMem : UDINT;
	_xInitOK : BOOL;
	_initState : _mntxt_initstate_enum;
	_CheckDoFunc : kgCheckDo;
	_CheckDoInst : kgCheckDo;
	_xInitDone : BOOL;
	_CheckDoPar : kgCheckDo;
	_CheckDoParHlp : kgCheckDo;
	_CheckDoMsg : kgCheckDo;
	_CheckDoMsgHlp : kgCheckDo;
END_VAR
```

### mnTxt_History.txt
```
0.03.0	02.01.12	AH	Texte werden nun eingelesen. Das Ändern der LCID bewirkt ein Neuladen der Texte
0.04.0	10.01.12	AH	PackageVersion wird in mnTxtStatAd angezeigt
0.04.1	12.01.12	AH	Ausgabe der korrekten Anzahl vorhandener Meldungs- und Meldungs-Hilfs-Zeilen
0.04.3	17.01.12	AH	Einlesen der Meldungs- und Meldungshilfstexte hat nicht funktioniert.
0.05.0	18.01.12	AH	Texte auf 63 Zeichen verlängert. Erfordert mnParam ab Version 0.10.0
0.06.0	17.02.12	AH  Speichernutzung optimiert
0.06.1	08.02.12	AH	Bugfix
0.07.0	13.03.12	AH	Datenobjektinitialisierung wieder in den Init-Teil gelegt
0.07.1	20.03.12	AH	Abhängigkeiten ergänzt
```

### Package Logical/Mewa/KGFramework/Pkg_hlDFII - DATAFOCUS II

### Pkg_hlDFII.typ - Global data types
```iecst
(********************************************************************
 * COPYRIGHT -- Microsoft
 ********************************************************************
 * Package: pkg_sqlreq
 * File: pkg_sqlreq.typ
 * Author: hunholz
 * Created: April 05, 2011
 ********************************************************************
 * Data types of package pkg_sqlreq
 ********************************************************************)

TYPE
	hlDFIIStatAd_typ : 	STRUCT
		sPkgVersion : STRING[10];
	END_STRUCT;
	hlDFIIParMac_typ : 	STRUCT
		bDBservReg : USINT := 3;
		bDBservAdr : USINT := 202;
		wDBservPort : UINT := 1433;
		sServInst : STRING[15];
		sDBname : STRING[15] := 'DFII';
		wIdletimeDisconnect : UINT := 10;
	END_STRUCT;
	hlDFIIPar_typ : 	STRUCT
		Mac : hlDFIIParMac_typ;
	END_STRUCT;
	IFhlDFII_typ : 	STRUCT
		In : IFhlDFII_In_typ;
		Out : IFhlDFII_Out_typ;
	END_STRUCT;
	IFhlDFII_Out_typ : 	STRUCT
		wStatus : UINT;
		xConnected : BOOL;
		RespProgByCat : IFhlDFII_Out_RespProgByCat_typ;
		RespMsgEvt : IFhlDFII_Out_RespMsgEvt_typ;
		RespCntBatchEvt : IFhlDFII_Out_RespCntBatchEvt_typ;
		RespCntCntEvt : IFhlDFII_Out_RespCntCntEvt_typ;
		RespCntTimEvt : IFhlDFII_Out_RespCntTimEvt_typ;
		RespCntDosEvt : IFhlDFII_Out_RespCntDosEvt_typ;
	END_STRUCT;
	IFhlDFII_In_typ : 	STRUCT
		utfMachineType : WSTRING[15];
		ReqProgByCat : IFhlDFII_In_ReqProgByCat_typ;
		ReqMsgEvt : IFhlDFII_In_ReqMsgEvt_typ;
		ReqCntBatchEvt : IFhlDFII_In_ReqCntBatchEvt_typ;
		ReqCntCntEvt : IFhlDFII_In_ReqCntCntEvt_typ;
		ReqCntTimEvt : IFhlDFII_In_ReqCntTimEvt_typ;
		ReqCntDosEvt : IFhlDFII_In_ReqCntDosEvt_typ;
	END_STRUCT;
	IFhlDFII_Out_RespProgByCat_typ : 	STRUCT
		wResponse : UINT; (*0 - idle, 1 - req num OK, 2 - req alpha OK, 65535 - busy*)
		bProgramNo : USINT;
		sProgramName : STRING[31];
		sCategoryName : STRING[31];
		wLoadrate : UINT;
		rSoilfactor : REAL;
		wColorIdxFor : UINT;
		wColorIdxBack : UINT;
	END_STRUCT;
	IFhlDFII_Out_RespMsgEvt_typ : 	STRUCT
		wResponse : UINT; (*0 - idle, 1 - req OK, 65535 - busy*)
	END_STRUCT;
	IFhlDFII_Out_RespCntBatchEvt_typ : 	STRUCT
		wResponse : UINT; (*0 - idle, 1 - req, OK, 65535 - busy*)
	END_STRUCT;
	IFhlDFII_Out_RespCntCntEvt_typ : 	STRUCT
		wResponse : UINT; (*0 - idle, 1 - req, OK, 65535 - busy*)
	END_STRUCT;
	IFhlDFII_Out_RespCntTimEvt_typ : 	STRUCT
		wResponse : UINT; (*0 - idle, 1 - req, OK, 65535 - busy*)
	END_STRUCT;
	IFhlDFII_Out_RespCntDosEvt_typ : 	STRUCT
		wResponse : UINT; (*0 - idle, 1 - req, OK, 65535 - busy*)
	END_STRUCT;
	IFhlDFII_In_ReqProgByCat_typ : 	STRUCT
		wRequest : UINT; (*0 - idle, 1 - req num, 2 - req alpha*)
		sCategoryNo_In : STRING[11];
	END_STRUCT;
	IFhlDFII_In_ReqMsgEvt_typ : 	STRUCT
		wRequest : UINT; (*0 - idle, 1 - req*)
		bCntLines : USINT; (*1..5*)
		MsgHistList : ARRAY[1..5]OF MsgHistList_Typ;
	END_STRUCT;
	IFhlDFII_In_ReqCntBatchEvt_typ : 	STRUCT
		wRequest : UINT; (*0 - idle, 1 - request*)
		bCntLines : USINT; (*1..5*)
		CntBatchEvtList : ARRAY[1..5]OF mnCntEventBatch_Typ;
	END_STRUCT;
	IFhlDFII_In_ReqCntCntEvt_typ : 	STRUCT
		wRequest : UINT; (*0 - idle, 1 - request*)
		bCntLines : USINT; (*1..5*)
		CntCounterEvtList : ARRAY[1..5]OF mnCntEventCounter_Typ;
	END_STRUCT;
	IFhlDFII_In_ReqCntTimEvt_typ : 	STRUCT
		wRequest : UINT; (*0 - idle, 1 - request*)
		bCntLines : USINT; (*1..5*)
		CntTimerEvtList : ARRAY[1..5]OF mnCntEventTime_Typ;
	END_STRUCT;
	IFhlDFII_In_ReqCntDosEvt_typ : 	STRUCT
		wRequest : UINT; (*0 - idle, 1 - request*)
		bCntLines : USINT; (*1..5*)
		CntDosingEvtList : ARRAY[1..5]OF mnCntEventDosingId_Typ;
	END_STRUCT;
END_TYPE
```

### Program Logical/Mewa/KGFramework/Pkg_hlDFII/hlDFII (IEC) - Statemachine zur Abfrage einer SQL-Datenbank
